LIN {X 0,Y 614.907,Z 968.972,A -85,B 0,C 180,E1 -6595.187,E2 -6595.187} C_VEL
LIN {X 0,Y 616.661,Z 950.759,A -85,B 0,C 180,E1 -6596.845,E2 -6596.845} C_VEL
LIN {X 0,Y 618.487,Z 931.255,A -85,B 0,C 180,E1 -6598.379,E2 -6598.379} C_VEL
LIN {X 0,Y 620.297,Z 912.013,A -85,B 0,C 180,E1 -6599.714,E2 -6599.714} C_VEL
LIN {X 0,Y 622.247,Z 890.482,A -85,B 0,C 180,E1 -6600.998,E2 -6600.998} C_VEL
LIN {X 0,Y 623.869,Z 871.366,A -85,B 0,C 180,E1 -6601.985,E2 -6601.985} C_VEL
LIN {X 0,Y 625.724,Z 847.82,A -85,B 0,C 180,E1 -6603.018,E2 -6603.018} C_VEL
LIN {X 0,Y 627.182,Z 825.971,A -85,B 0,C 180,E1 -6603.807,E2 -6603.807} C_VEL
LIN {X 0,Y 628.648,Z 801.827,A -85,B 0,C 180,E1 -6604.51,E2 -6604.51} C_VEL
LIN {X 0,Y 629.71,Z 779.15,A -85,B 0,C 180,E1 -6605.003,E2 -6605.003} C_VEL
LIN {X 0,Y 630.482,Z 755.478,A -85,B 0,C 180,E1 -6605.381,E2 -6605.381} C_VEL
LIN {X 0,Y 634.576,Z 507.829,A -85,B 0,C 180,E1 -6608.538,E2 -6608.538} C_VEL
LIN {X 0,Y 636.13,Z 410.472,A -85,B 0,C 180,E1 -6609.804,E2 -6609.804} C_VEL
LIN {X 0,Y 632.258,Z 394.616,A -85,B 0,C 180,E1 -6610.318,E2 -6610.318} C_VEL
LIN {X 0,Y 620.448,Z 374.384,A -85,B 0,C 180,E1 -6611.533,E2 -6611.533} C_VEL
LIN {X 0,Y 612.728,Z 354.981,A -85,B 0,C 180,E1 -6613.911,E2 -6613.911} C_VEL
LIN {X 0,Y 609.065,Z 345.367,A -85,B 0,C 180,E1 -6615.133,E2 -6615.133} C_VEL
LIN {X 0,Y 609.009,Z 345.37,A -85,B 0,C 180,E1 -6618.07,E2 -6618.07} C_VEL
LIN {X 0,Y 609.077,Z 345.362,A -85,B 0,C 180,E1 -6621.163,E2 -6621.163} C_VEL
LIN {X 0,Y 609.012,Z 345.368,A -85,B 0,C 180,E1 -6624.233,E2 -6624.233} C_VEL
LIN {X 0,Y 609.057,Z 345.366,A -85,B 0,C 180,E1 -6627.42,E2 -6627.42} C_VEL
LIN {X 0,Y 609.014,Z 345.363,A -85,B 0,C 180,E1 -6630.384,E2 -6630.384} C_VEL
LIN {X 0,Y 609.062,Z 345.353,A -85,B 0,C 180,E1 -6633.478,E2 -6633.478} C_VEL
LIN {X 0,Y 609.009,Z 345.353,A -85,B 0,C 180,E1 -6636.384,E2 -6636.384} C_VEL
LIN {X 0,Y 609.076,Z 345.362,A -85,B 0,C 180,E1 -6639.432,E2 -6639.432} C_VEL
LIN {X 0,Y 609.011,Z 345.364,A -85,B 0,C 180,E1 -6642.515,E2 -6642.515} C_VEL
LIN {X 0,Y 609.07,Z 345.348,A -85,B 0,C 180,E1 -6645.647,E2 -6645.647} C_VEL
LIN {X 0,Y 609.012,Z 345.364,A -85,B 0,C 180,E1 -6648.637,E2 -6648.637} C_VEL
LIN {X 0,Y 609.064,Z 345.355,A -85,B 0,C 180,E1 -6651.789,E2 -6651.789} C_VEL
LIN {X 0,Y 609.012,Z 345.356,A -85,B 0,C 180,E1 -6654.725,E2 -6654.725} C_VEL
LIN {X 0,Y 609.069,Z 345.364,A -85,B 0,C 180,E1 -6657.836,E2 -6657.836} C_VEL
LIN {X 0,Y 609.011,Z 345.346,A -85,B 0,C 180,E1 -6660.847,E2 -6660.847} C_VEL
LIN {X 0,Y 609.068,Z 345.363,A -85,B 0,C 180,E1 -6663.954,E2 -6663.954} C_VEL
LIN {X 0,Y 609.014,Z 345.357,A -85,B 0,C 180,E1 -6666.978,E2 -6666.978} C_VEL
LIN {X 0,Y 609.06,Z 345.352,A -85,B 0,C 180,E1 -6670.117,E2 -6670.117} C_VEL
LIN {X 0,Y 609.016,Z 345.364,A -85,B 0,C 180,E1 -6673.095,E2 -6673.095} C_VEL
LIN {X 0,Y 609.062,Z 345.349,A -85,B 0,C 180,E1 -6676.206,E2 -6676.206} C_VEL
LIN {X 0,Y 609.017,Z 345.363,A -85,B 0,C 180,E1 -6679.17,E2 -6679.17} C_VEL
LIN {X 0,Y 609.072,Z 345.357,A -85,B 0,C 180,E1 -6682.286,E2 -6682.286} C_VEL
LIN {X 0,Y 609.013,Z 345.35,A -85,B 0,C 180,E1 -6685.269,E2 -6685.269} C_VEL
LIN {X 0,Y 609.064,Z 345.357,A -85,B 0,C 180,E1 -6688.43,E2 -6688.43} C_VEL
LIN {X 0,Y 609.017,Z 345.366,A -85,B 0,C 180,E1 -6691.379,E2 -6691.379} C_VEL
LIN {X 0,Y 609.065,Z 345.36,A -85,B 0,C 180,E1 -6694.5,E2 -6694.5} C_VEL
LIN {X 0,Y 609.018,Z 345.364,A -85,B 0,C 180,E1 -6697.534,E2 -6697.534} C_VEL
LIN {X 0,Y 609.061,Z 345.36,A -85,B 0,C 180,E1 -6700.674,E2 -6700.674} C_VEL
LIN {X 0,Y 609.015,Z 345.332,A -85,B 0,C 180,E1 -6703.611,E2 -6703.611} C_VEL
LIN {X 0,Y 609.059,Z 345.368,A -85,B 0,C 180,E1 -6706.797,E2 -6706.797} C_VEL
LIN {X 0,Y 609.062,Z 345.576,A -85,B 0,C 180,E1 -6709.113,E2 -6709.113} C_VEL
LIN {X 0,Y 611.013,Z 350.763,A -85,B 0,C 180,E1 -6709.765,E2 -6709.765} C_VEL
LIN {X 0,Y 626.828,Z 375.591,A -85,B 0,C 180,E1 -6711.41,E2 -6711.41} C_VEL
LIN {X 0,Y 636.341,Z 391.797,A -85,B 0,C 180,E1 -6712.363,E2 -6712.363} C_VEL
LIN {X 0,Y 635.973,Z 412.733,A -85,B 0,C 180,E1 -6712.635,E2 -6712.635} C_VEL
LIN {X 0,Y 635.046,Z 420.434,A -85,B 0,C 180,E1 -6712.677,E2 -6712.677} C_VEL
LIN {X 0,Y 629.809,Z 441.007,A -85,B 0,C 180,E1 -6712.587,E2 -6712.587} C_VEL
LIN {X 0,Y 629.133,Z 447.61,A -85,B 0,C 180,E1 -6712.632,E2 -6712.632} C_VEL
LIN {X 0,Y 624.626,Z 698.687,A -85,B 0,C 180,E1 -6715.87,E2 -6715.87} C_VEL
LIN {X 0,Y 623.697,Z 743.497,A -85,B 0,C 180,E1 -6716.476,E2 -6716.476} C_VEL
LIN {X 0,Y 622.627,Z 767.01,A -85,B 0,C 180,E1 -6716.956,E2 -6716.956} C_VEL
LIN {X 0,Y 621.497,Z 787.189,A -85,B 0,C 180,E1 -6717.49,E2 -6717.49} C_VEL
LIN {X 0,Y 619.803,Z 812.008,A -85,B 0,C 180,E1 -6718.324,E2 -6718.324} C_VEL
LIN {X 0,Y 618.178,Z 832.167,A -85,B 0,C 180,E1 -6719.153,E2 -6719.153} C_VEL
LIN {X 0,Y 616.198,Z 855.203,A -85,B 0,C 180,E1 -6720.282,E2 -6720.282} C_VEL
LIN {X 0,Y 614.304,Z 874.686,A -85,B 0,C 180,E1 -6721.41,E2 -6721.41} C_VEL
LIN {X 0,Y 612.292,Z 894.753,A -85,B 0,C 180,E1 -6722.738,E2 -6722.738} C_VEL
LIN {X 0,Y 610.169,Z 914.461,A -85,B 0,C 180,E1 -6724.262,E2 -6724.262} C_VEL
LIN {X 0,Y 608.261,Z 932.973,A -85,B 0,C 180,E1 -6725.89,E2 -6725.89} C_VEL
LIN {X 0,Y 606.372,Z 950.537,A -85,B 0,C 180,E1 -6727.68,E2 -6727.68} C_VEL
LIN {X 0,Y 604.843,Z 966.182,A -85,B 0,C 180,E1 -6729.484,E2 -6729.484} C_VEL
LIN {X 0,Y 603.374,Z 981.698,A -85,B 0,C 180,E1 -6731.548,E2 -6731.548} C_VEL
LIN {X 0,Y 602.275,Z 995.359,A -85,B 0,C 180,E1 -6733.607,E2 -6733.607} C_VEL
LIN {X 0,Y 601.407,Z 1007.51,A -85,B 0,C 180,E1 -6735.764,E2 -6735.764} C_VEL
LIN {X 0,Y 600.8,Z 1017.904,A -85,B 0,C 180,E1 -6737.895,E2 -6737.895} C_VEL
LIN {X 0,Y 600.376,Z 1026.879,A -85,B 0,C 180,E1 -6740.123,E2 -6740.123} C_VEL
LIN {X 0,Y 600.123,Z 1033.674,A -85,B 0,C 180,E1 -6742.148,E2 -6742.148} C_VEL
LIN {X 0,Y 599.975,Z 1040.012,A -85,B 0,C 180,E1 -6744.549,E2 -6744.549} C_VEL
LIN {X 0,Y 599.921,Z 1043.917,A -85,B 0,C 180,E1 -6746.56,E2 -6746.56} C_VEL
LIN {X 0,Y 599.913,Z 1046.869,A -85,B 0,C 180,E1 -6748.758,E2 -6748.758} C_VEL
LIN {X 0,Y 599.909,Z 1048.271,A -85,B 0,C 180,E1 -6751.051,E2 -6751.051} C_VEL
LIN {X 0,Y 599.907,Z 1048.267,A -85,B 0,C 180,E1 -6753.057,E2 -6753.057} C_VEL
LIN {X 0,Y 599.914,Z 1046.729,A -85,B 0,C 180,E1 -6755.452,E2 -6755.452} C_VEL
LIN {X 0,Y 599.92,Z 1043.857,A -85,B 0,C 180,E1 -6757.566,E2 -6757.566} C_VEL
LIN {X 0,Y 599.977,Z 1039.899,A -85,B 0,C 180,E1 -6759.593,E2 -6759.593} C_VEL
LIN {X 0,Y 600.131,Z 1033.43,A -85,B 0,C 180,E1 -6762.021,E2 -6762.021} C_VEL
LIN {X 0,Y 600.376,Z 1026.855,A -85,B 0,C 180,E1 -6763.974,E2 -6763.974} C_VEL
LIN {X 0,Y 600.809,Z 1017.709,A -85,B 0,C 180,E1 -6766.236,E2 -6766.236} C_VEL
LIN {X 0,Y 601.404,Z 1007.563,A -85,B 0,C 180,E1 -6768.314,E2 -6768.314} C_VEL
LIN {X 0,Y 602.235,Z 995.823,A -85,B 0,C 180,E1 -6770.406,E2 -6770.406} C_VEL
LIN {X 0,Y 603.299,Z 982.647,A -85,B 0,C 180,E1 -6772.408,E2 -6772.408} C_VEL
LIN {X 0,Y 604.779,Z 966.914,A -85,B 0,C 180,E1 -6774.518,E2 -6774.518} C_VEL
LIN {X 0,Y 606.352,Z 950.764,A -85,B 0,C 180,E1 -6776.386,E2 -6776.386} C_VEL
LIN {X 0,Y 608.209,Z 933.493,A -85,B 0,C 180,E1 -6778.153,E2 -6778.153} C_VEL
LIN {X 0,Y 610.106,Z 915.133,A -85,B 0,C 180,E1 -6779.774,E2 -6779.774} C_VEL
LIN {X 0,Y 612.122,Z 896.309,A -85,B 0,C 180,E1 -6781.24,E2 -6781.24} C_VEL
LIN {X 0,Y 614.194,Z 875.91,A -85,B 0,C 180,E1 -6782.606,E2 -6782.606} C_VEL
LIN {X 0,Y 615.954,Z 857.768,A -85,B 0,C 180,E1 -6783.667,E2 -6783.667} C_VEL
LIN {X 0,Y 617.994,Z 834.601,A -85,B 0,C 180,E1 -6784.83,E2 -6784.83} C_VEL
LIN {X 0,Y 619.641,Z 814.117,A -85,B 0,C 180,E1 -6785.686,E2 -6785.686} C_VEL
LIN {X 0,Y 621.334,Z 790.192,A -85,B 0,C 180,E1 -6786.514,E2 -6786.514} C_VEL
LIN {X 0,Y 622.573,Z 768.29,A -85,B 0,C 180,E1 -6787.105,E2 -6787.105} C_VEL
LIN {X 0,Y 623.558,Z 746.916,A -85,B 0,C 180,E1 -6787.553,E2 -6787.553} C_VEL
LIN {X 0,Y 624.385,Z 714.088,A -85,B 0,C 180,E1 -6788.027,E2 -6788.027} C_VEL
LIN {X 0,Y 629.115,Z 459.765,A -85,B 0,C 180,E1 -6791.323,E2 -6791.323} C_VEL
LIN {X 0,Y 630.263,Z 394.469,A -85,B 0,C 180,E1 -6792.193,E2 -6792.193} C_VEL
LIN {X 0,Y 616.493,Z 371.695,A -85,B 0,C 180,E1 -6793.666,E2 -6793.666} C_VEL
LIN {X 0,Y 604.629,Z 353.842,A -85,B 0,C 180,E1 -6794.994,E2 -6794.994} C_VEL
LIN {X 0,Y 602.702,Z 350.561,A -85,B 0,C 180,E1 -6795.24,E2 -6795.24} C_VEL
LIN {X 0,Y 601.12,Z 346.347,A -85,B 0,C 180,E1 -6795.859,E2 -6795.859} C_VEL
LIN {X 0,Y 601.072,Z 346.326,A -85,B 0,C 180,E1 -6798.795,E2 -6798.795} C_VEL
LIN {X 0,Y 601.127,Z 346.352,A -85,B 0,C 180,E1 -6801.895,E2 -6801.895} C_VEL
LIN {X 0,Y 601.077,Z 346.322,A -85,B 0,C 180,E1 -6804.977,E2 -6804.977} C_VEL
LIN {X 0,Y 601.104,Z 346.343,A -85,B 0,C 180,E1 -6808.213,E2 -6808.213} C_VEL
LIN {X 0,Y 601.084,Z 346.351,A -85,B 0,C 180,E1 -6811.157,E2 -6811.157} C_VEL
LIN {X 0,Y 601.088,Z 346.344,A -85,B 0,C 180,E1 -6814.479,E2 -6814.479} C_VEL
LIN {X 0,Y 601.096,Z 346.355,A -85,B 0,C 180,E1 -6817.402,E2 -6817.402} C_VEL
LIN {X 0,Y 601.083,Z 346.353,A -85,B 0,C 180,E1 -6820.668,E2 -6820.668} C_VEL
LIN {X 0,Y 601.113,Z 346.353,A -85,B 0,C 180,E1 -6823.695,E2 -6823.695} C_VEL
LIN {X 0,Y 601.078,Z 346.349,A -85,B 0,C 180,E1 -6826.827,E2 -6826.827} C_VEL
LIN {X 0,Y 601.116,Z 346.343,A -85,B 0,C 180,E1 -6829.844,E2 -6829.844} C_VEL
LIN {X 0,Y 601.076,Z 346.352,A -85,B 0,C 180,E1 -6833.025,E2 -6833.025} C_VEL
LIN {X 0,Y 601.13,Z 346.353,A -85,B 0,C 180,E1 -6836.09,E2 -6836.09} C_VEL
LIN {X 0,Y 601.071,Z 346.345,A -85,B 0,C 180,E1 -6839.237,E2 -6839.237} C_VEL
LIN {X 0,Y 601.135,Z 346.339,A -85,B 0,C 180,E1 -6842.288,E2 -6842.288} C_VEL
LIN {X 0,Y 601.072,Z 346.355,A -85,B 0,C 180,E1 -6845.441,E2 -6845.441} C_VEL
LIN {X 0,Y 601.14,Z 346.35,A -85,B 0,C 180,E1 -6848.513,E2 -6848.513} C_VEL
LIN {X 0,Y 601.071,Z 346.34,A -85,B 0,C 180,E1 -6851.612,E2 -6851.612} C_VEL
LIN {X 0,Y 601.132,Z 346.337,A -85,B 0,C 180,E1 -6854.744,E2 -6854.744} C_VEL
LIN {X 0,Y 601.076,Z 346.355,A -85,B 0,C 180,E1 -6857.823,E2 -6857.823} C_VEL
LIN {X 0,Y 601.107,Z 346.352,A -85,B 0,C 180,E1 -6861.065,E2 -6861.065} C_VEL
LIN {X 0,Y 601.074,Z 346.344,A -85,B 0,C 180,E1 -6863.947,E2 -6863.947} C_VEL
LIN {X 0,Y 601.108,Z 346.341,A -85,B 0,C 180,E1 -6867.136,E2 -6867.136} C_VEL
LIN {X 0,Y 601.078,Z 346.354,A -85,B 0,C 180,E1 -6870.047,E2 -6870.047} C_VEL
LIN {X 0,Y 601.103,Z 346.355,A -85,B 0,C 180,E1 -6873.294,E2 -6873.294} C_VEL
LIN {X 0,Y 601.079,Z 346.357,A -85,B 0,C 180,E1 -6876.216,E2 -6876.216} C_VEL
LIN {X 0,Y 601.093,Z 346.355,A -85,B 0,C 180,E1 -6879.48,E2 -6879.48} C_VEL
LIN {X 0,Y 601.079,Z 346.346,A -85,B 0,C 180,E1 -6882.355,E2 -6882.355} C_VEL
LIN {X 0,Y 601.088,Z 346.48,A -85,B 0,C 180,E1 -6883.997,E2 -6883.997} C_VEL
LIN {X 0,Y 602.408,Z 349.863,A -85,B 0,C 180,E1 -6884.463,E2 -6884.463} C_VEL
LIN {X 0,Y 610.096,Z 368.505,A -85,B 0,C 180,E1 -6886.967,E2 -6886.967} C_VEL
LIN {X 0,Y 612.618,Z 374.622,A -85,B 0,C 180,E1 -6887.713,E2 -6887.713} C_VEL
LIN {X 0,Y 626.907,Z 398.785,A -85,B 0,C 180,E1 -6889.271,E2 -6889.271} C_VEL
LIN {X 0,Y 630.302,Z 413.187,A -85,B 0,C 180,E1 -6889.753,E2 -6889.753} C_VEL
LIN {X 0,Y 625.305,Z 678.851,A -85,B 0,C 180,E1 -6893.209,E2 -6893.209} C_VEL
LIN {X 0,Y 623.609,Z 766.876,A -85,B 0,C 180,E1 -6894.36,E2 -6894.36} C_VEL
LIN {X 0,Y 622.513,Z 792.116,A -85,B 0,C 180,E1 -6894.847,E2 -6894.847} C_VEL
LIN {X 0,Y 621.327,Z 812.813,A -85,B 0,C 180,E1 -6895.38,E2 -6895.38} C_VEL
LIN {X 0,Y 619.815,Z 835.949,A -85,B 0,C 180,E1 -6896.126,E2 -6896.126} C_VEL
LIN {X 0,Y 618.029,Z 858.133,A -85,B 0,C 180,E1 -6897.015,E2 -6897.015} C_VEL
LIN {X 0,Y 616.219,Z 879.499,A -85,B 0,C 180,E1 -6898.026,E2 -6898.026} C_VEL
LIN {X 0,Y 614.165,Z 901.367,A -85,B 0,C 180,E1 -6899.256,E2 -6899.256} C_VEL
LIN {X 0,Y 612.36,Z 919.919,A -85,B 0,C 180,E1 -6900.454,E2 -6900.454} C_VEL
LIN {X 0,Y 610.169,Z 941.37,A -85,B 0,C 180,E1 -6902.052,E2 -6902.052} C_VEL
LIN {X 0,Y 608.466,Z 958.204,A -85,B 0,C 180,E1 -6903.488,E2 -6903.488} C_VEL
LIN {X 0,Y 606.561,Z 977.386,A -85,B 0,C 180,E1 -6905.351,E2 -6905.351} C_VEL
LIN {X 0,Y 605.093,Z 992.65,A -85,B 0,C 180,E1 -6907.047,E2 -6907.047} C_VEL
LIN {X 0,Y 603.751,Z 1007.707,A -85,B 0,C 180,E1 -6908.938,E2 -6908.938} C_VEL
LIN {X 0,Y 602.589,Z 1021.238,A -85,B 0,C 180,E1 -6910.92,E2 -6910.92} C_VEL
LIN {X 0,Y 601.668,Z 1033.688,A -85,B 0,C 180,E1 -6912.993,E2 -6912.993} C_VEL
LIN {X 0,Y 600.962,Z 1044.707,A -85,B 0,C 180,E1 -6915.168,E2 -6915.168} C_VEL
LIN {X 0,Y 600.515,Z 1053.583,A -85,B 0,C 180,E1 -6917.206,E2 -6917.206} C_VEL
LIN {X 0,Y 600.189,Z 1061.907,A -85,B 0,C 180,E1 -6919.538,E2 -6919.538} C_VEL
LIN {X 0,Y 600.028,Z 1067.491,A -85,B 0,C 180,E1 -6921.471,E2 -6921.471} C_VEL
LIN {X 0,Y 599.946,Z 1072.695,A -85,B 0,C 180,E1 -6923.781,E2 -6923.781} C_VEL
LIN {X 0,Y 599.911,Z 1076.009,A -85,B 0,C 180,E1 -6925.986,E2 -6925.986} C_VEL
LIN {X 0,Y 599.906,Z 1077.835,A -85,B 0,C 180,E1 -6927.994,E2 -6927.994} C_VEL
LIN {X 0,Y 599.895,Z 1078.417,A -85,B 0,C 180,E1 -6930.382,E2 -6930.382} C_VEL
LIN {X 0,Y 599.908,Z 1077.495,A -85,B 0,C 180,E1 -6932.484,E2 -6932.484} C_VEL
LIN {X 0,Y 599.925,Z 1075.085,A -85,B 0,C 180,E1 -6934.78,E2 -6934.78} C_VEL
LIN {X 0,Y 599.968,Z 1071.102,A -85,B 0,C 180,E1 -6936.988,E2 -6936.988} C_VEL
LIN {X 0,Y 600.05,Z 1066.219,A -85,B 0,C 180,E1 -6939.012,E2 -6939.012} C_VEL
LIN {X 0,Y 600.302,Z 1058.66,A -85,B 0,C 180,E1 -6941.432,E2 -6941.432} C_VEL
LIN {X 0,Y 600.649,Z 1050.747,A -85,B 0,C 180,E1 -6943.477,E2 -6943.477} C_VEL
LIN {X 0,Y 601.23,Z 1040.401,A -85,B 0,C 180,E1 -6945.729,E2 -6945.729} C_VEL
LIN {X 0,Y 601.991,Z 1029.111,A -85,B 0,C 180,E1 -6947.795,E2 -6947.795} C_VEL
LIN {X 0,Y 603.057,Z 1015.705,A -85,B 0,C 180,E1 -6949.93,E2 -6949.93} C_VEL
LIN {X 0,Y 604.209,Z 1002.366,A -85,B 0,C 180,E1 -6951.758,E2 -6951.758} C_VEL
LIN {X 0,Y 605.684,Z 986.675,A -85,B 0,C 180,E1 -6953.65,E2 -6953.65} C_VEL
LIN {X 0,Y 607.335,Z 969.481,A -85,B 0,C 180,E1 -6955.448,E2 -6955.448} C_VEL
LIN {X 0,Y 609.031,Z 952.779,A -85,B 0,C 180,E1 -6956.997,E2 -6956.997} C_VEL
LIN {X 0,Y 611.099,Z 932.382,A -85,B 0,C 180,E1 -6958.647,E2 -6958.647} C_VEL
LIN {X 0,Y 612.926,Z 914.014,A -85,B 0,C 180,E1 -6959.946,E2 -6959.946} C_VEL
LIN {X 0,Y 615.152,Z 891.169,A -85,B 0,C 180,E1 -6961.342,E2 -6961.342} C_VEL
LIN {X 0,Y 616.861,Z 872.159,A -85,B 0,C 180,E1 -6962.338,E2 -6962.338} C_VEL
LIN {X 0,Y 618.757,Z 849.985,A -85,B 0,C 180,E1 -6963.336,E2 -6963.336} C_VEL
LIN {X 0,Y 620.364,Z 827.239,A -85,B 0,C 180,E1 -6964.174,E2 -6964.174} C_VEL
LIN {X 0,Y 621.869,Z 804.051,A -85,B 0,C 180,E1 -6964.869,E2 -6964.869} C_VEL
LIN {X 0,Y 623.087,Z 780.045,A -85,B 0,C 180,E1 -6965.406,E2 -6965.406} C_VEL
LIN {X 0,Y 623.869,Z 757.754,A -85,B 0,C 180,E1 -6965.771,E2 -6965.771} C_VEL
LIN {X 0,Y 628.139,Z 514.362,A -85,B 0,C 180,E1 -6968.903,E2 -6968.903} C_VEL
LIN {X 0,Y 629.865,Z 412.184,A -85,B 0,C 180,E1 -6970.243,E2 -6970.243} C_VEL
LIN {X 0,Y 626.549,Z 398.688,A -85,B 0,C 180,E1 -6970.691,E2 -6970.691} C_VEL
LIN {X 0,Y 612.132,Z 374.17,A -85,B 0,C 180,E1 -6972.202,E2 -6972.202} C_VEL
LIN {X 0,Y 605.013,Z 356.379,A -85,B 0,C 180,E1 -6974.442,E2 -6974.442} C_VEL
LIN {X 0,Y 602.095,Z 349.342,A -85,B 0,C 180,E1 -6975.374,E2 -6975.374} C_VEL
LIN {X 0,Y 601.073,Z 346.362,A -85,B 0,C 180,E1 -6975.782,E2 -6975.782} C_VEL
LIN {X 0,Y 601.141,Z 346.354,A -85,B 0,C 180,E1 -6978.893,E2 -6978.893} C_VEL
LIN {X 0,Y 601.072,Z 346.354,A -85,B 0,C 180,E1 -6982.012,E2 -6982.012} C_VEL
LIN {X 0,Y 601.137,Z 346.344,A -85,B 0,C 180,E1 -6985.097,E2 -6985.097} C_VEL
LIN {X 0,Y 601.07,Z 346.351,A -85,B 0,C 180,E1 -6988.174,E2 -6988.174} C_VEL
LIN {X 0,Y 601.146,Z 346.349,A -85,B 0,C 180,E1 -6991.269,E2 -6991.269} C_VEL
LIN {X 0,Y 601.073,Z 346.353,A -85,B 0,C 180,E1 -6994.373,E2 -6994.373} C_VEL
LIN {X 0,Y 601.128,Z 346.34,A -85,B 0,C 180,E1 -6997.507,E2 -6997.507} C_VEL
LIN {X 0,Y 601.071,Z 346.344,A -85,B 0,C 180,E1 -7000.466,E2 -7000.466} C_VEL
LIN {X 0,Y 601.132,Z 346.354,A -85,B 0,C 180,E1 -7003.574,E2 -7003.574} C_VEL
LIN {X 0,Y 601.071,Z 346.348,A -85,B 0,C 180,E1 -7006.533,E2 -7006.533} C_VEL
LIN {X 0,Y 601.13,Z 346.339,A -85,B 0,C 180,E1 -7009.651,E2 -7009.651} C_VEL
LIN {X 0,Y 601.073,Z 346.354,A -85,B 0,C 180,E1 -7012.641,E2 -7012.641} C_VEL
LIN {X 0,Y 601.132,Z 346.334,A -85,B 0,C 180,E1 -7015.707,E2 -7015.707} C_VEL
LIN {X 0,Y 601.073,Z 346.353,A -85,B 0,C 180,E1 -7018.763,E2 -7018.763} C_VEL
LIN {X 0,Y 601.129,Z 346.339,A -85,B 0,C 180,E1 -7021.906,E2 -7021.906} C_VEL
LIN {X 0,Y 601.075,Z 346.346,A -85,B 0,C 180,E1 -7024.962,E2 -7024.962} C_VEL
LIN {X 0,Y 601.119,Z 346.354,A -85,B 0,C 180,E1 -7028.128,E2 -7028.128} C_VEL
LIN {X 0,Y 601.077,Z 346.335,A -85,B 0,C 180,E1 -7031.126,E2 -7031.126} C_VEL
LIN {X 0,Y 601.106,Z 346.351,A -85,B 0,C 180,E1 -7034.35,E2 -7034.35} C_VEL
LIN {X 0,Y 601.084,Z 346.347,A -85,B 0,C 180,E1 -7037.323,E2 -7037.323} C_VEL
LIN {X 0,Y 601.087,Z 346.339,A -85,B 0,C 180,E1 -7040.65,E2 -7040.65} C_VEL
LIN {X 0,Y 601.096,Z 346.353,A -85,B 0,C 180,E1 -7043.572,E2 -7043.572} C_VEL
LIN {X 0,Y 601.088,Z 346.357,A -85,B 0,C 180,E1 -7046.795,E2 -7046.795} C_VEL
LIN {X 0,Y 601.101,Z 346.337,A -85,B 0,C 180,E1 -7049.737,E2 -7049.737} C_VEL
LIN {X 0,Y 601.083,Z 346.343,A -85,B 0,C 180,E1 -7052.954,E2 -7052.954} C_VEL
LIN {X 0,Y 601.115,Z 346.351,A -85,B 0,C 180,E1 -7055.957,E2 -7055.957} C_VEL
LIN {X 0,Y 601.079,Z 346.351,A -85,B 0,C 180,E1 -7059.178,E2 -7059.178} C_VEL
LIN {X 0,Y 601.133,Z 346.345,A -85,B 0,C 180,E1 -7062.221,E2 -7062.221} C_VEL
LIN {X 0,Y 601.073,Z 346.328,A -85,B 0,C 180,E1 -7065.397,E2 -7065.397} C_VEL
LIN {X 0,Y 601.153,Z 346.432,A -85,B 0,C 180,E1 -7068.487,E2 -7068.487} C_VEL
LIN {X 0,Y 602.862,Z 351.065,A -85,B 0,C 180,E1 -7069.076,E2 -7069.076} C_VEL
LIN {X 0,Y 616.619,Z 372.529,A -85,B 0,C 180,E1 -7070.559,E2 -7070.559} C_VEL
LIN {X 0,Y 630.095,Z 394.837,A -85,B 0,C 180,E1 -7071.941,E2 -7071.941} C_VEL
LIN {X 0,Y 629.133,Z 447.61,A -85,B 0,C 180,E1 -7072.632,E2 -7072.632} C_VEL
LIN {X 0,Y 628.244,Z 455.305,A -85,B 0,C 180,E1 -7072.677,E2 -7072.677} C_VEL
LIN {X 0,Y 622.959,Z 475.868,A -85,B 0,C 180,E1 -7072.583,E2 -7072.583} C_VEL
LIN {X 0,Y 622.23,Z 482.476,A -85,B 0,C 180,E1 -7072.624,E2 -7072.624} C_VEL
LIN {X 0,Y 617.517,Z 731.007,A -85,B 0,C 180,E1 -7075.856,E2 -7075.856} C_VEL
LIN {X 0,Y 616.722,Z 753.294,A -85,B 0,C 180,E1 -7076.227,E2 -7076.227} C_VEL
LIN {X 0,Y 615.459,Z 777.86,A -85,B 0,C 180,E1 -7076.792,E2 -7076.792} C_VEL
LIN {X 0,Y 614.004,Z 799.911,A -85,B 0,C 180,E1 -7077.466,E2 -7077.466} C_VEL
LIN {X 0,Y 612.299,Z 822.879,A -85,B 0,C 180,E1 -7078.325,E2 -7078.325} C_VEL
LIN {X 0,Y 610.303,Z 844.777,A -85,B 0,C 180,E1 -7079.332,E2 -7079.332} C_VEL
LIN {X 0,Y 608.392,Z 864.519,A -85,B 0,C 180,E1 -7080.391,E2 -7080.391} C_VEL
LIN {X 0,Y 606.038,Z 886.679,A -85,B 0,C 180,E1 -7081.786,E2 -7081.786} C_VEL
LIN {X 0,Y 604.102,Z 904.459,A -85,B 0,C 180,E1 -7083.077,E2 -7083.077} C_VEL
LIN {X 0,Y 601.738,Z 925.356,A -85,B 0,C 180,E1 -7084.825,E2 -7084.825} C_VEL
LIN {X 0,Y 599.882,Z 941.946,A -85,B 0,C 180,E1 -7086.42,E2 -7086.42} C_VEL
LIN {X 0,Y 597.901,Z 960.025,A -85,B 0,C 180,E1 -7088.413,E2 -7088.413} C_VEL
LIN {X 0,Y 596.425,Z 974.226,A -85,B 0,C 180,E1 -7090.206,E2 -7090.206} C_VEL
LIN {X 0,Y 594.973,Z 989.307,A -85,B 0,C 180,E1 -7092.392,E2 -7092.392} C_VEL
LIN {X 0,Y 593.962,Z 1001.792,A -85,B 0,C 180,E1 -7094.475,E2 -7094.475} C_VEL
LIN {X 0,Y 593.142,Z 1013.486,A -85,B 0,C 180,E1 -7096.746,E2 -7096.746} C_VEL
LIN {X 0,Y 592.636,Z 1022.096,A -85,B 0,C 180,E1 -7098.714,E2 -7098.714} C_VEL
LIN {X 0,Y 592.261,Z 1030.49,A -85,B 0,C 180,E1 -7100.982,E2 -7100.982} C_VEL
LIN {X 0,Y 592.049,Z 1036.745,A -85,B 0,C 180,E1 -7103.113,E2 -7103.113} C_VEL
LIN {X 0,Y 591.963,Z 1041.511,A -85,B 0,C 180,E1 -7105.155,E2 -7105.155} C_VEL
LIN {X 0,Y 591.923,Z 1045.542,A -85,B 0,C 180,E1 -7107.58,E2 -7107.58} C_VEL
LIN {X 0,Y 591.905,Z 1047.554,A -85,B 0,C 180,E1 -7109.613,E2 -7109.613} C_VEL
LIN {X 0,Y 591.896,Z 1048.437,A -85,B 0,C 180,E1 -7111.742,E2 -7111.742} C_VEL
LIN {X 0,Y 591.913,Z 1047.773,A -85,B 0,C 180,E1 -7114.166,E2 -7114.166} C_VEL
LIN {X 0,Y 591.922,Z 1045.899,A -85,B 0,C 180,E1 -7116.206,E2 -7116.206} C_VEL
LIN {X 0,Y 591.95,Z 1042.329,A -85,B 0,C 180,E1 -7118.548,E2 -7118.548} C_VEL
LIN {X 0,Y 592.038,Z 1037.192,A -85,B 0,C 180,E1 -7120.805,E2 -7120.805} C_VEL
LIN {X 0,Y 592.239,Z 1031.206,A -85,B 0,C 180,E1 -7122.877,E2 -7122.877} C_VEL
LIN {X 0,Y 592.617,Z 1022.571,A -85,B 0,C 180,E1 -7125.261,E2 -7125.261} C_VEL
LIN {X 0,Y 593.118,Z 1013.869,A -85,B 0,C 180,E1 -7127.26,E2 -7127.26} C_VEL
LIN {X 0,Y 593.945,Z 1002.028,A -85,B 0,C 180,E1 -7129.573,E2 -7129.573} C_VEL
LIN {X 0,Y 594.974,Z 989.301,A -85,B 0,C 180,E1 -7131.699,E2 -7131.699} C_VEL
LIN {X 0,Y 596.458,Z 973.859,A -85,B 0,C 180,E1 -7133.934,E2 -7133.934} C_VEL
LIN {X 0,Y 597.891,Z 960.118,A -85,B 0,C 180,E1 -7135.667,E2 -7135.667} C_VEL
LIN {X 0,Y 599.873,Z 942.069,A -85,B 0,C 180,E1 -7137.659,E2 -7137.659} C_VEL
LIN {X 0,Y 601.647,Z 926.152,A -85,B 0,C 180,E1 -7139.194,E2 -7139.194} C_VEL
LIN {X 0,Y 603.862,Z 906.891,A -85,B 0,C 180,E1 -7140.829,E2 -7140.829} C_VEL
LIN {X 0,Y 605.902,Z 888.072,A -85,B 0,C 180,E1 -7142.21,E2 -7142.21} C_VEL
LIN {X 0,Y 608.117,Z 867.448,A -85,B 0,C 180,E1 -7143.536,E2 -7143.536} C_VEL
LIN {X 0,Y 610.217,Z 845.785,A -85,B 0,C 180,E1 -7144.709,E2 -7144.709} C_VEL
LIN {X 0,Y 612.113,Z 825.036,A -85,B 0,C 180,E1 -7145.673,E2 -7145.673} C_VEL
LIN {X 0,Y 613.912,Z 801.822,A -85,B 0,C 180,E1 -7146.563,E2 -7146.563} C_VEL
LIN {X 0,Y 615.308,Z 781.023,A -85,B 0,C 180,E1 -7147.213,E2 -7147.213} C_VEL
LIN {X 0,Y 616.707,Z 754.929,A -85,B 0,C 180,E1 -7147.84,E2 -7147.84} C_VEL
LIN {X 0,Y 617.54,Z 732.814,A -85,B 0,C 180,E1 -7148.218,E2 -7148.218} C_VEL
LIN {X 0,Y 622.498,Z 483.595,A -85,B 0,C 180,E1 -7151.483,E2 -7151.483} C_VEL
LIN {X 0,Y 624.172,Z 397.807,A -85,B 0,C 180,E1 -7152.63,E2 -7152.63} C_VEL
LIN {X 0,Y 611.713,Z 377.111,A -85,B 0,C 180,E1 -7153.993,E2 -7153.993} C_VEL
LIN {X 0,Y 600.335,Z 359.822,A -85,B 0,C 180,E1 -7155.292,E2 -7155.292} C_VEL
LIN {X 0,Y 594.515,Z 350.884,A -85,B 0,C 180,E1 -7156.004,E2 -7156.004} C_VEL
LIN {X 0,Y 593.137,Z 347.34,A -85,B 0,C 180,E1 -7156.544,E2 -7156.544} C_VEL
LIN {X 0,Y 593.201,Z 347.303,A -85,B 0,C 180,E1 -7159.664,E2 -7159.664} C_VEL
LIN {X 0,Y 593.135,Z 347.329,A -85,B 0,C 180,E1 -7162.757,E2 -7162.757} C_VEL
LIN {X 0,Y 593.186,Z 347.326,A -85,B 0,C 180,E1 -7165.97,E2 -7165.97} C_VEL
LIN {X 0,Y 593.138,Z 347.336,A -85,B 0,C 180,E1 -7168.946,E2 -7168.946} C_VEL
LIN {X 0,Y 593.191,Z 347.334,A -85,B 0,C 180,E1 -7172.056,E2 -7172.056} C_VEL
LIN {X 0,Y 593.139,Z 347.334,A -85,B 0,C 180,E1 -7175.086,E2 -7175.086} C_VEL
LIN {X 0,Y 593.169,Z 347.33,A -85,B 0,C 180,E1 -7178.336,E2 -7178.336} C_VEL
LIN {X 0,Y 593.146,Z 347.342,A -85,B 0,C 180,E1 -7181.331,E2 -7181.331} C_VEL
LIN {X 0,Y 593.148,Z 347.34,A -85,B 0,C 180,E1 -7184.653,E2 -7184.653} C_VEL
LIN {X 0,Y 593.152,Z 347.341,A -85,B 0,C 180,E1 -7187.539,E2 -7187.539} C_VEL
LIN {X 0,Y 593.14,Z 347.337,A -85,B 0,C 180,E1 -7190.882,E2 -7190.882} C_VEL
LIN {X 0,Y 593.166,Z 347.334,A -85,B 0,C 180,E1 -7193.807,E2 -7193.807} C_VEL
LIN {X 0,Y 593.139,Z 347.342,A -85,B 0,C 180,E1 -7197.004,E2 -7197.004} C_VEL
LIN {X 0,Y 593.177,Z 347.337,A -85,B 0,C 180,E1 -7200,E2 -7200} C_VEL
LIN {X 0,Y 593.135,Z 347.331,A -85,B 0,C 180,E1 -7203.189,E2 -7203.189} C_VEL
LIN {X 0,Y 593.195,Z 347.329,A -85,B 0,C 180,E1 -7206.29,E2 -7206.29} C_VEL
LIN {X 0,Y 593.134,Z 347.344,A -85,B 0,C 180,E1 -7209.411,E2 -7209.411} C_VEL
LIN {X 0,Y 593.199,Z 347.336,A -85,B 0,C 180,E1 -7212.59,E2 -7212.59} C_VEL
LIN {X 0,Y 593.131,Z 347.329,A -85,B 0,C 180,E1 -7215.648,E2 -7215.648} C_VEL
LIN {X 0,Y 593.191,Z 347.325,A -85,B 0,C 180,E1 -7218.781,E2 -7218.781} C_VEL
LIN {X 0,Y 593.135,Z 347.345,A -85,B 0,C 180,E1 -7221.873,E2 -7221.873} C_VEL
LIN {X 0,Y 593.178,Z 347.341,A -85,B 0,C 180,E1 -7225.03,E2 -7225.03} C_VEL
LIN {X 0,Y 593.139,Z 347.339,A -85,B 0,C 180,E1 -7228.056,E2 -7228.056} C_VEL
LIN {X 0,Y 593.16,Z 347.342,A -85,B 0,C 180,E1 -7231.279,E2 -7231.279} C_VEL
LIN {X 0,Y 593.146,Z 347.348,A -85,B 0,C 180,E1 -7234.266,E2 -7234.266} C_VEL
LIN {X 0,Y 593.142,Z 347.343,A -85,B 0,C 180,E1 -7237.607,E2 -7237.607} C_VEL
LIN {X 0,Y 593.157,Z 347.344,A -85,B 0,C 180,E1 -7240.513,E2 -7240.513} C_VEL
LIN {X 0,Y 593.203,Z 347.514,A -85,B 0,C 180,E1 -7243.317,E2 -7243.317} C_VEL
LIN {X 0,Y 594.313,Z 350.62,A -85,B 0,C 180,E1 -7243.748,E2 -7243.748} C_VEL
LIN {X 0,Y 599.743,Z 363.46,A -85,B 0,C 180,E1 -7245.555,E2 -7245.555} C_VEL
LIN {X 0,Y 604.178,Z 374.241,A -85,B 0,C 180,E1 -7246.96,E2 -7246.96} C_VEL
LIN {X 0,Y 615.048,Z 392.088,A -85,B 0,C 180,E1 -7248.193,E2 -7248.193} C_VEL
LIN {X 0,Y 621.799,Z 403.971,A -85,B 0,C 180,E1 -7248.937,E2 -7248.937} C_VEL
LIN {X 0,Y 624.187,Z 415.618,A -85,B 0,C 180,E1 -7249.305,E2 -7249.305} C_VEL
LIN {X 0,Y 618.894,Z 680.404,A -85,B 0,C 180,E1 -7252.782,E2 -7252.782} C_VEL
LIN {X 0,Y 617.125,Z 766.737,A -85,B 0,C 180,E1 -7253.923,E2 -7253.923} C_VEL
LIN {X 0,Y 615.96,Z 791.941,A -85,B 0,C 180,E1 -7254.413,E2 -7254.413} C_VEL
LIN {X 0,Y 614.692,Z 812.825,A -85,B 0,C 180,E1 -7254.956,E2 -7254.956} C_VEL
LIN {X 0,Y 612.984,Z 837.056,A -85,B 0,C 180,E1 -7255.753,E2 -7255.753} C_VEL
LIN {X 0,Y 611.217,Z 857.916,A -85,B 0,C 180,E1 -7256.6,E2 -7256.6} C_VEL
LIN {X 0,Y 609.321,Z 878.967,A -85,B 0,C 180,E1 -7257.603,E2 -7257.603} C_VEL
LIN {X 0,Y 607.109,Z 901.141,A -85,B 0,C 180,E1 -7258.859,E2 -7258.859} C_VEL
LIN {X 0,Y 605.152,Z 920.171,A -85,B 0,C 180,E1 -7260.102,E2 -7260.102} C_VEL
LIN {X 0,Y 602.881,Z 941.145,A -85,B 0,C 180,E1 -7261.684,E2 -7261.684} C_VEL
LIN {X 0,Y 601.038,Z 958.14,A -85,B 0,C 180,E1 -7263.149,E2 -7263.149} C_VEL
LIN {X 0,Y 599.032,Z 977.16,A -85,B 0,C 180,E1 -7265.02,E2 -7265.02} C_VEL
LIN {X 0,Y 597.458,Z 992.425,A -85,B 0,C 180,E1 -7266.736,E2 -7266.736} C_VEL
LIN {X 0,Y 595.961,Z 1008.237,A -85,B 0,C 180,E1 -7268.752,E2 -7268.752} C_VEL
LIN {X 0,Y 594.797,Z 1021.223,A -85,B 0,C 180,E1 -7270.66,E2 -7270.66} C_VEL
LIN {X 0,Y 593.816,Z 1033.688,A -85,B 0,C 180,E1 -7272.761,E2 -7272.761} C_VEL
LIN {X 0,Y 593.06,Z 1044.637,A -85,B 0,C 180,E1 -7274.951,E2 -7274.951} C_VEL
LIN {X 0,Y 592.57,Z 1053.582,A -85,B 0,C 180,E1 -7277.031,E2 -7277.031} C_VEL
LIN {X 0,Y 592.22,Z 1061.907,A -85,B 0,C 180,E1 -7279.395,E2 -7279.395} C_VEL
LIN {X 0,Y 592.033,Z 1067.745,A -85,B 0,C 180,E1 -7281.453,E2 -7281.453} C_VEL
LIN {X 0,Y 591.947,Z 1073.015,A -85,B 0,C 180,E1 -7283.891,E2 -7283.891} C_VEL
LIN {X 0,Y 591.912,Z 1076.008,A -85,B 0,C 180,E1 -7285.932,E2 -7285.932} C_VEL
LIN {X 0,Y 591.907,Z 1077.835,A -85,B 0,C 180,E1 -7287.967,E2 -7287.967} C_VEL
LIN {X 0,Y 591.895,Z 1078.417,A -85,B 0,C 180,E1 -7290.387,E2 -7290.387} C_VEL
LIN {X 0,Y 591.907,Z 1077.494,A -85,B 0,C 180,E1 -7292.517,E2 -7292.517} C_VEL
LIN {X 0,Y 591.928,Z 1075.085,A -85,B 0,C 180,E1 -7294.845,E2 -7294.845} C_VEL
LIN {X 0,Y 591.98,Z 1071.102,A -85,B 0,C 180,E1 -7297.083,E2 -7297.083} C_VEL
LIN {X 0,Y 592.069,Z 1066.219,A -85,B 0,C 180,E1 -7299.134,E2 -7299.134} C_VEL
LIN {X 0,Y 592.341,Z 1058.659,A -85,B 0,C 180,E1 -7301.588,E2 -7301.588} C_VEL
LIN {X 0,Y 592.713,Z 1050.747,A -85,B 0,C 180,E1 -7303.661,E2 -7303.661} C_VEL
LIN {X 0,Y 593.342,Z 1040.4,A -85,B 0,C 180,E1 -7305.943,E2 -7305.943} C_VEL
LIN {X 0,Y 594.115,Z 1029.683,A -85,B 0,C 180,E1 -7307.938,E2 -7307.938} C_VEL
LIN {X 0,Y 595.078,Z 1018.012,A -85,B 0,C 180,E1 -7309.841,E2 -7309.841} C_VEL
LIN {X 0,Y 596.44,Z 1002.925,A -85,B 0,C 180,E1 -7311.953,E2 -7311.953} C_VEL
LIN {X 0,Y 597.812,Z 989.017,A -85,B 0,C 180,E1 -7313.667,E2 -7313.667} C_VEL
LIN {X 0,Y 599.748,Z 970.285,A -85,B 0,C 180,E1 -7315.688,E2 -7315.688} C_VEL
LIN {X 0,Y 601.538,Z 953.68,A -85,B 0,C 180,E1 -7317.254,E2 -7317.254} C_VEL
LIN {X 0,Y 603.791,Z 932.835,A -85,B 0,C 180,E1 -7318.972,E2 -7318.972} C_VEL
LIN {X 0,Y 605.723,Z 914.534,A -85,B 0,C 180,E1 -7320.285,E2 -7320.285} C_VEL
LIN {X 0,Y 608.081,Z 891.856,A -85,B 0,C 180,E1 -7321.693,E2 -7321.693} C_VEL
LIN {X 0,Y 609.97,Z 871.941,A -85,B 0,C 180,E1 -7322.748,E2 -7322.748} C_VEL
LIN {X 0,Y 611.957,Z 849.956,A -85,B 0,C 180,E1 -7323.747,E2 -7323.747} C_VEL
LIN {X 0,Y 613.666,Z 826.975,A -85,B 0,C 180,E1 -7324.599,E2 -7324.599} C_VEL
LIN {X 0,Y 615.272,Z 803.625,A -85,B 0,C 180,E1 -7325.302,E2 -7325.302} C_VEL
LIN {X 0,Y 616.529,Z 779.786,A -85,B 0,C 180,E1 -7325.836,E2 -7325.836} C_VEL
LIN {X 0,Y 617.343,Z 757.549,A -85,B 0,C 180,E1 -7326.203,E2 -7326.203} C_VEL
LIN {X 0,Y 621.875,Z 513.243,A -85,B 0,C 180,E1 -7329.374,E2 -7329.374} C_VEL
LIN {X 0,Y 623.645,Z 413.984,A -85,B 0,C 180,E1 -7330.689,E2 -7330.689} C_VEL
LIN {X 0,Y 620.948,Z 402.893,A -85,B 0,C 180,E1 -7331.061,E2 -7331.061} C_VEL
LIN {X 0,Y 606.513,Z 378.526,A -85,B 0,C 180,E1 -7332.6,E2 -7332.6} C_VEL
LIN {X 0,Y 603.652,Z 373.695,A -85,B 0,C 180,E1 -7332.934,E2 -7332.934} C_VEL
LIN {X 0,Y 596.249,Z 354.957,A -85,B 0,C 180,E1 -7335.36,E2 -7335.36} C_VEL
LIN {X 0,Y 593.174,Z 347.515,A -85,B 0,C 180,E1 -7336.38,E2 -7336.38} C_VEL
LIN {X 0,Y 593.143,Z 347.338,A -85,B 0,C 180,E1 -7339.659,E2 -7339.659} C_VEL
LIN {X 0,Y 593.154,Z 347.335,A -85,B 0,C 180,E1 -7342.558,E2 -7342.558} C_VEL
LIN {X 0,Y 593.137,Z 347.335,A -85,B 0,C 180,E1 -7345.864,E2 -7345.864} C_VEL
LIN {X 0,Y 593.179,Z 347.329,A -85,B 0,C 180,E1 -7348.905,E2 -7348.905} C_VEL
LIN {X 0,Y 593.135,Z 347.333,A -85,B 0,C 180,E1 -7352.054,E2 -7352.054} C_VEL
LIN {X 0,Y 593.198,Z 347.34,A -85,B 0,C 180,E1 -7355.183,E2 -7355.183} C_VEL
LIN {X 0,Y 593.132,Z 347.344,A -85,B 0,C 180,E1 -7358.259,E2 -7358.259} C_VEL
LIN {X 0,Y 593.196,Z 347.323,A -85,B 0,C 180,E1 -7361.321,E2 -7361.321} C_VEL
LIN {X 0,Y 593.133,Z 347.338,A -85,B 0,C 180,E1 -7364.452,E2 -7364.452} C_VEL
LIN {X 0,Y 593.199,Z 347.337,A -85,B 0,C 180,E1 -7367.54,E2 -7367.54} C_VEL
LIN {X 0,Y 593.134,Z 347.325,A -85,B 0,C 180,E1 -7370.687,E2 -7370.687} C_VEL
LIN {X 0,Y 593.176,Z 347.337,A -85,B 0,C 180,E1 -7373.904,E2 -7373.904} C_VEL
LIN {X 0,Y 593.139,Z 347.337,A -85,B 0,C 180,E1 -7376.908,E2 -7376.908} C_VEL
LIN {X 0,Y 593.156,Z 347.324,A -85,B 0,C 180,E1 -7380.193,E2 -7380.193} C_VEL
LIN {X 0,Y 593.152,Z 347.341,A -85,B 0,C 180,E1 -7383.189,E2 -7383.189} C_VEL
LIN {X 0,Y 593.142,Z 347.33,A -85,B 0,C 180,E1 -7386.485,E2 -7386.485} C_VEL
LIN {X 0,Y 593.174,Z 347.34,A -85,B 0,C 180,E1 -7389.509,E2 -7389.509} C_VEL
LIN {X 0,Y 593.138,Z 347.343,A -85,B 0,C 180,E1 -7392.758,E2 -7392.758} C_VEL
LIN {X 0,Y 593.189,Z 347.326,A -85,B 0,C 180,E1 -7395.747,E2 -7395.747} C_VEL
LIN {X 0,Y 593.138,Z 347.343,A -85,B 0,C 180,E1 -7398.885,E2 -7398.885} C_VEL
LIN {X 0,Y 593.203,Z 347.327,A -85,B 0,C 180,E1 -7402.018,E2 -7402.018} C_VEL
LIN {X 0,Y 593.136,Z 347.327,A -85,B 0,C 180,E1 -7405.142,E2 -7405.142} C_VEL
LIN {X 0,Y 593.203,Z 347.335,A -85,B 0,C 180,E1 -7408.272,E2 -7408.272} C_VEL
LIN {X 0,Y 593.138,Z 347.344,A -85,B 0,C 180,E1 -7411.28,E2 -7411.28} C_VEL
LIN {X 0,Y 593.196,Z 347.333,A -85,B 0,C 180,E1 -7414.38,E2 -7414.38} C_VEL
LIN {X 0,Y 593.139,Z 347.342,A -85,B 0,C 180,E1 -7417.486,E2 -7417.486} C_VEL
LIN {X 0,Y 593.184,Z 347.337,A -85,B 0,C 180,E1 -7420.665,E2 -7420.665} C_VEL
LIN {X 0,Y 593.142,Z 347.303,A -85,B 0,C 180,E1 -7423.722,E2 -7423.722} C_VEL
LIN {X 0,Y 593.154,Z 347.344,A -85,B 0,C 180,E1 -7427.076,E2 -7427.076} C_VEL
LIN {X 0,Y 593.154,Z 347.392,A -85,B 0,C 180,E1 -7427.839,E2 -7427.839} C_VEL
LIN {X 0,Y 594.654,Z 351.038,A -85,B 0,C 180,E1 -7428.349,E2 -7428.349} C_VEL
LIN {X 0,Y 597.659,Z 355.727,A -85,B 0,C 180,E1 -7428.693,E2 -7428.693} C_VEL
LIN {X 0,Y 614.201,Z 381.749,A -85,B 0,C 180,E1 -7430.503,E2 -7430.503} C_VEL
LIN {X 0,Y 623.877,Z 398.119,A -85,B 0,C 180,E1 -7431.514,E2 -7431.514} C_VEL
LIN {X 0,Y 622.23,Z 482.476,A -85,B 0,C 180,E1 -7432.624,E2 -7432.624} C_VEL
LIN {X 0,Y 621.294,Z 490.172,A -85,B 0,C 180,E1 -7432.667,E2 -7432.667} C_VEL
LIN {X 0,Y 616.01,Z 510.726,A -85,B 0,C 180,E1 -7432.571,E2 -7432.571} C_VEL
LIN {X 0,Y 615.282,Z 517.33,A -85,B 0,C 180,E1 -7432.613,E2 -7432.613} C_VEL
LIN {X 0,Y 610.798,Z 738.818,A -85,B 0,C 180,E1 -7435.53,E2 -7435.53} C_VEL
LIN {X 0,Y 609.666,Z 764.83,A -85,B 0,C 180,E1 -7436.034,E2 -7436.034} C_VEL
LIN {X 0,Y 608.431,Z 785.229,A -85,B 0,C 180,E1 -7436.568,E2 -7436.568} C_VEL
LIN {X 0,Y 606.832,Z 808.119,A -85,B 0,C 180,E1 -7437.316,E2 -7437.316} C_VEL
LIN {X 0,Y 604.856,Z 830.468,A -85,B 0,C 180,E1 -7438.23,E2 -7438.23} C_VEL
LIN {X 0,Y 602.904,Z 851.104,A -85,B 0,C 180,E1 -7439.227,E2 -7439.227} C_VEL
LIN {X 0,Y 600.587,Z 872.854,A -85,B 0,C 180,E1 -7440.475,E2 -7440.475} C_VEL
LIN {X 0,Y 598.536,Z 891.142,A -85,B 0,C 180,E1 -7441.689,E2 -7441.689} C_VEL
LIN {X 0,Y 596.051,Z 912.338,A -85,B 0,C 180,E1 -7443.313,E2 -7443.313} C_VEL
LIN {X 0,Y 594.016,Z 929.15,A -85,B 0,C 180,E1 -7444.794,E2 -7444.794} C_VEL
LIN {X 0,Y 591.899,Z 947.25,A -85,B 0,C 180,E1 -7446.61,E2 -7446.61} C_VEL
LIN {X 0,Y 590.061,Z 962.964,A -85,B 0,C 180,E1 -7448.425,E2 -7448.425} C_VEL
LIN {X 0,Y 588.41,Z 978.342,A -85,B 0,C 180,E1 -7450.442,E2 -7450.442} C_VEL
LIN {X 0,Y 587.046,Z 991.568,A -85,B 0,C 180,E1 -7452.454,E2 -7452.454} C_VEL
LIN {X 0,Y 585.976,Z 1003.957,A -85,B 0,C 180,E1 -7454.602,E2 -7454.602} C_VEL
LIN {X 0,Y 585.111,Z 1015.437,A -85,B 0,C 180,E1 -7456.963,E2 -7456.963} C_VEL
LIN {X 0,Y 584.562,Z 1024.976,A -85,B 0,C 180,E1 -7459.255,E2 -7459.255} C_VEL
LIN {X 0,Y 584.217,Z 1032.642,A -85,B 0,C 180,E1 -7461.536,E2 -7461.536} C_VEL
LIN {X 0,Y 584.029,Z 1038.844,A -85,B 0,C 180,E1 -7463.808,E2 -7463.808} C_VEL
LIN {X 0,Y 583.939,Z 1043.53,A -85,B 0,C 180,E1 -7466.171,E2 -7466.171} C_VEL
LIN {X 0,Y 583.916,Z 1046.369,A -85,B 0,C 180,E1 -7468.234,E2 -7468.234} C_VEL
LIN {X 0,Y 583.905,Z 1048.193,A -85,B 0,C 180,E1 -7470.687,E2 -7470.687} C_VEL
LIN {X 0,Y 583.901,Z 1048.322,A -85,B 0,C 180,E1 -7472.847,E2 -7472.847} C_VEL
LIN {X 0,Y 583.907,Z 1047.208,A -85,B 0,C 180,E1 -7475.01,E2 -7475.01} C_VEL
LIN {X 0,Y 583.921,Z 1044.246,A -85,B 0,C 180,E1 -7477.478,E2 -7477.478} C_VEL
LIN {X 0,Y 583.981,Z 1040.488,A -85,B 0,C 180,E1 -7479.519,E2 -7479.519} C_VEL
LIN {X 0,Y 584.138,Z 1034.778,A -85,B 0,C 180,E1 -7481.853,E2 -7481.853} C_VEL
LIN {X 0,Y 584.42,Z 1027.715,A -85,B 0,C 180,E1 -7484.061,E2 -7484.061} C_VEL
LIN {X 0,Y 584.85,Z 1019.591,A -85,B 0,C 180,E1 -7486.181,E2 -7486.181} C_VEL
LIN {X 0,Y 585.612,Z 1008.323,A -85,B 0,C 180,E1 -7488.62,E2 -7488.62} C_VEL
LIN {X 0,Y 586.517,Z 997.396,A -85,B 0,C 180,E1 -7490.664,E2 -7490.664} C_VEL
LIN {X 0,Y 587.799,Z 983.988,A -85,B 0,C 180,E1 -7492.82,E2 -7492.82} C_VEL
LIN {X 0,Y 589.206,Z 970.769,A -85,B 0,C 180,E1 -7494.675,E2 -7494.675} C_VEL
LIN {X 0,Y 591.158,Z 953.447,A -85,B 0,C 180,E1 -7496.793,E2 -7496.793} C_VEL
LIN {X 0,Y 592.998,Z 937.922,A -85,B 0,C 180,E1 -7498.447,E2 -7498.447} C_VEL
LIN {X 0,Y 595.316,Z 918.528,A -85,B 0,C 180,E1 -7500.257,E2 -7500.257} C_VEL
LIN {X 0,Y 597.342,Z 901.341,A -85,B 0,C 180,E1 -7501.653,E2 -7501.653} C_VEL
LIN {X 0,Y 599.727,Z 881.124,A -85,B 0,C 180,E1 -7503.094,E2 -7503.094} C_VEL
LIN {X 0,Y 601.926,Z 860.711,A -85,B 0,C 180,E1 -7504.336,E2 -7504.336} C_VEL
LIN {X 0,Y 604.066,Z 839.682,A -85,B 0,C 180,E1 -7505.446,E2 -7505.446} C_VEL
LIN {X 0,Y 606.1,Z 817.103,A -85,B 0,C 180,E1 -7506.434,E2 -7506.434} C_VEL
LIN {X 0,Y 607.771,Z 795.967,A -85,B 0,C 180,E1 -7507.206,E2 -7507.206} C_VEL
LIN {X 0,Y 609.436,Z 771.119,A -85,B 0,C 180,E1 -7507.921,E2 -7507.921} C_VEL
LIN {X 0,Y 610.501,Z 750.521,A -85,B 0,C 180,E1 -7508.373,E2 -7508.373} C_VEL
LIN {X 0,Y 611.38,Z 724.593,A -85,B 0,C 180,E1 -7508.786,E2 -7508.786} C_VEL
LIN {X 0,Y 616.669,Z 471.349,A -85,B 0,C 180,E1 -7512.128,E2 -7512.128} C_VEL
LIN {X 0,Y 618.093,Z 401.034,A -85,B 0,C 180,E1 -7513.08,E2 -7513.08} C_VEL
LIN {X 0,Y 606.633,Z 382.039,A -85,B 0,C 180,E1 -7514.362,E2 -7514.362} C_VEL
LIN {X 0,Y 596.058,Z 365.802,A -85,B 0,C 180,E1 -7515.594,E2 -7515.594} C_VEL
LIN {X 0,Y 589.397,Z 356.043,A -85,B 0,C 180,E1 -7516.4,E2 -7516.4} C_VEL
LIN {X 0,Y 586.094,Z 351.126,A -85,B 0,C 180,E1 -7516.834,E2 -7516.834} C_VEL
LIN {X 0,Y 585.241,Z 348.333,A -85,B 0,C 180,E1 -7517.278,E2 -7517.278} C_VEL
LIN {X 0,Y 585.198,Z 348.309,A -85,B 0,C 180,E1 -7520.407,E2 -7520.407} C_VEL
LIN {X 0,Y 585.238,Z 348.294,A -85,B 0,C 180,E1 -7523.418,E2 -7523.418} C_VEL
LIN {X 0,Y 585.198,Z 348.333,A -85,B 0,C 180,E1 -7526.62,E2 -7526.62} C_VEL
LIN {X 0,Y 585.268,Z 348.331,A -85,B 0,C 180,E1 -7529.822,E2 -7529.822} C_VEL
LIN {X 0,Y 585.199,Z 348.333,A -85,B 0,C 180,E1 -7532.967,E2 -7532.967} C_VEL
LIN {X 0,Y 585.239,Z 348.331,A -85,B 0,C 180,E1 -7536.221,E2 -7536.221} C_VEL
LIN {X 0,Y 585.201,Z 348.325,A -85,B 0,C 180,E1 -7539.182,E2 -7539.182} C_VEL
LIN {X 0,Y 585.225,Z 348.321,A -85,B 0,C 180,E1 -7542.435,E2 -7542.435} C_VEL
LIN {X 0,Y 585.208,Z 348.326,A -85,B 0,C 180,E1 -7545.453,E2 -7545.453} C_VEL
LIN {X 0,Y 585.207,Z 348.329,A -85,B 0,C 180,E1 -7548.768,E2 -7548.768} C_VEL
LIN {X 0,Y 585.236,Z 348.33,A -85,B 0,C 180,E1 -7551.847,E2 -7551.847} C_VEL
LIN {X 0,Y 585.199,Z 348.324,A -85,B 0,C 180,E1 -7555.001,E2 -7555.001} C_VEL
LIN {X 0,Y 585.252,Z 348.316,A -85,B 0,C 180,E1 -7558.14,E2 -7558.14} C_VEL
LIN {X 0,Y 585.195,Z 348.333,A -85,B 0,C 180,E1 -7561.273,E2 -7561.273} C_VEL
LIN {X 0,Y 585.258,Z 348.329,A -85,B 0,C 180,E1 -7564.409,E2 -7564.409} C_VEL
LIN {X 0,Y 585.192,Z 348.317,A -85,B 0,C 180,E1 -7567.461,E2 -7567.461} C_VEL
LIN {X 0,Y 585.251,Z 348.315,A -85,B 0,C 180,E1 -7570.633,E2 -7570.633} C_VEL
LIN {X 0,Y 585.197,Z 348.334,A -85,B 0,C 180,E1 -7573.739,E2 -7573.739} C_VEL
LIN {X 0,Y 585.229,Z 348.33,A -85,B 0,C 180,E1 -7576.987,E2 -7576.987} C_VEL
LIN {X 0,Y 585.203,Z 348.318,A -85,B 0,C 180,E1 -7579.992,E2 -7579.992} C_VEL
LIN {X 0,Y 585.204,Z 348.317,A -85,B 0,C 180,E1 -7583.353,E2 -7583.353} C_VEL
LIN {X 0,Y 585.229,Z 348.323,A -85,B 0,C 180,E1 -7586.374,E2 -7586.374} C_VEL
LIN {X 0,Y 585.2,Z 348.331,A -85,B 0,C 180,E1 -7589.59,E2 -7589.59} C_VEL
LIN {X 0,Y 585.249,Z 348.331,A -85,B 0,C 180,E1 -7592.676,E2 -7592.676} C_VEL
LIN {X 0,Y 585.194,Z 348.336,A -85,B 0,C 180,E1 -7595.879,E2 -7595.879} C_VEL
LIN {X 0,Y 585.26,Z 348.328,A -85,B 0,C 180,E1 -7599.081,E2 -7599.081} C_VEL
LIN {X 0,Y 585.194,Z 348.326,A -85,B 0,C 180,E1 -7602.136,E2 -7602.136} C_VEL
LIN {X 0,Y 585.223,Z 348.344,A -85,B 0,C 180,E1 -7602.578,E2 -7602.578} C_VEL
LIN {X 0,Y 586.681,Z 351.97,A -85,B 0,C 180,E1 -7603.113,E2 -7603.113} C_VEL
LIN {X 0,Y 593.473,Z 368.351,A -85,B 0,C 180,E1 -7605.453,E2 -7605.453} C_VEL
LIN {X 0,Y 595.931,Z 373.949,A -85,B 0,C 180,E1 -7606.195,E2 -7606.195} C_VEL
LIN {X 0,Y 609.554,Z 396.18,A -85,B 0,C 180,E1 -7607.785,E2 -7607.785} C_VEL
LIN {X 0,Y 616.287,Z 408.139,A -85,B 0,C 180,E1 -7608.545,E2 -7608.545} C_VEL
LIN {X 0,Y 618.126,Z 417.453,A -85,B 0,C 180,E1 -7608.84,E2 -7608.84} C_VEL
LIN {X 0,Y 612.536,Z 681.518,A -85,B 0,C 180,E1 -7612.339,E2 -7612.339} C_VEL
LIN {X 0,Y 610.689,Z 766.523,A -85,B 0,C 180,E1 -7613.474,E2 -7613.474} C_VEL
LIN {X 0,Y 609.446,Z 791.914,A -85,B 0,C 180,E1 -7613.971,E2 -7613.971} C_VEL
LIN {X 0,Y 608.087,Z 813.136,A -85,B 0,C 180,E1 -7614.529,E2 -7614.529} C_VEL
LIN {X 0,Y 606.241,Z 837.672,A -85,B 0,C 180,E1 -7615.35,E2 -7615.35} C_VEL
LIN {X 0,Y 604.447,Z 857.777,A -85,B 0,C 180,E1 -7616.176,E2 -7616.176} C_VEL
LIN {X 0,Y 602.438,Z 878.777,A -85,B 0,C 180,E1 -7617.187,E2 -7617.187} C_VEL
LIN {X 0,Y 600.086,Z 900.917,A -85,B 0,C 180,E1 -7618.453,E2 -7618.453} C_VEL
LIN {X 0,Y 597.986,Z 920.207,A -85,B 0,C 180,E1 -7619.726,E2 -7619.726} C_VEL
LIN {X 0,Y 595.62,Z 940.919,A -85,B 0,C 180,E1 -7621.307,E2 -7621.307} C_VEL
LIN {X 0,Y 593.657,Z 957.901,A -85,B 0,C 180,E1 -7622.787,E2 -7622.787} C_VEL
LIN {X 0,Y 591.447,Z 977.584,A -85,B 0,C 180,E1 -7624.752,E2 -7624.752} C_VEL
LIN {X 0,Y 589.845,Z 992.199,A -85,B 0,C 180,E1 -7626.418,E2 -7626.418} C_VEL
LIN {X 0,Y 588.248,Z 1008.013,A -85,B 0,C 180,E1 -7628.46,E2 -7628.46} C_VEL
LIN {X 0,Y 586.994,Z 1020.999,A -85,B 0,C 180,E1 -7630.393,E2 -7630.393} C_VEL
LIN {X 0,Y 585.964,Z 1033.662,A -85,B 0,C 180,E1 -7632.532,E2 -7632.532} C_VEL
LIN {X 0,Y 585.19,Z 1044.177,A -85,B 0,C 180,E1 -7634.642,E2 -7634.642} C_VEL
LIN {X 0,Y 584.663,Z 1052.897,A -85,B 0,C 180,E1 -7636.683,E2 -7636.683} C_VEL
LIN {X 0,Y 584.256,Z 1061.604,A -85,B 0,C 180,E1 -7639.149,E2 -7639.149} C_VEL
LIN {X 0,Y 584.044,Z 1067.491,A -85,B 0,C 180,E1 -7641.236,E2 -7641.236} C_VEL
LIN {X 0,Y 583.946,Z 1072.695,A -85,B 0,C 180,E1 -7643.61,E2 -7643.61} C_VEL
LIN {X 0,Y 583.915,Z 1075.894,A -85,B 0,C 180,E1 -7645.777,E2 -7645.777} C_VEL
LIN {X 0,Y 583.909,Z 1077.766,A -85,B 0,C 180,E1 -7647.841,E2 -7647.841} C_VEL
LIN {X 0,Y 583.898,Z 1078.439,A -85,B 0,C 180,E1 -7650.294,E2 -7650.294} C_VEL
LIN {X 0,Y 583.908,Z 1077.562,A -85,B 0,C 180,E1 -7652.454,E2 -7652.454} C_VEL
LIN {X 0,Y 583.922,Z 1075.439,A -85,B 0,C 180,E1 -7654.616,E2 -7654.616} C_VEL
LIN {X 0,Y 583.982,Z 1071.308,A -85,B 0,C 180,E1 -7657.081,E2 -7657.081} C_VEL
LIN {X 0,Y 584.077,Z 1066.474,A -85,B 0,C 180,E1 -7659.161,E2 -7659.161} C_VEL
LIN {X 0,Y 584.348,Z 1059.365,A -85,B 0,C 180,E1 -7661.549,E2 -7661.549} C_VEL
LIN {X 0,Y 584.735,Z 1051.556,A -85,B 0,C 180,E1 -7663.649,E2 -7663.649} C_VEL
LIN {X 0,Y 585.357,Z 1041.888,A -85,B 0,C 180,E1 -7665.861,E2 -7665.861} C_VEL
LIN {X 0,Y 586.229,Z 1030.138,A -85,B 0,C 180,E1 -7668.085,E2 -7668.085} C_VEL
LIN {X 0,Y 587.241,Z 1018.436,A -85,B 0,C 180,E1 -7670.013,E2 -7670.013} C_VEL
LIN {X 0,Y 588.68,Z 1003.484,A -85,B 0,C 180,E1 -7672.152,E2 -7672.152} C_VEL
LIN {X 0,Y 590.127,Z 989.651,A -85,B 0,C 180,E1 -7673.888,E2 -7673.888} C_VEL
LIN {X 0,Y 592.068,Z 972.111,A -85,B 0,C 180,E1 -7675.831,E2 -7675.831} C_VEL
LIN {X 0,Y 593.989,Z 955.14,A -85,B 0,C 180,E1 -7677.467,E2 -7677.467} C_VEL
LIN {X 0,Y 596.231,Z 935.921,A -85,B 0,C 180,E1 -7679.105,E2 -7679.105} C_VEL
LIN {X 0,Y 598.376,Z 916.536,A -85,B 0,C 180,E1 -7680.53,E2 -7680.53} C_VEL
LIN {X 0,Y 600.66,Z 896.054,A -85,B 0,C 180,E1 -7681.85,E2 -7681.85} C_VEL
LIN {X 0,Y 602.819,Z 874.727,A -85,B 0,C 180,E1 -7683.016,E2 -7683.016} C_VEL
LIN {X 0,Y 604.633,Z 855.575,A -85,B 0,C 180,E1 -7683.917,E2 -7683.917} C_VEL
LIN {X 0,Y 606.634,Z 831.946,A -85,B 0,C 180,E1 -7684.853,E2 -7684.853} C_VEL
LIN {X 0,Y 608.207,Z 809.82,A -85,B 0,C 180,E1 -7685.555,E2 -7685.555} C_VEL
LIN {X 0,Y 609.71,Z 785.451,A -85,B 0,C 180,E1 -7686.162,E2 -7686.162} C_VEL
LIN {X 0,Y 610.708,Z 761.524,A -85,B 0,C 180,E1 -7686.581,E2 -7686.581} C_VEL
LIN {X 0,Y 615.333,Z 527.23,A -85,B 0,C 180,E1 -7689.656,E2 -7689.656} C_VEL
LIN {X 0,Y 617.477,Z 415.813,A -85,B 0,C 180,E1 -7691.141,E2 -7691.141} C_VEL
LIN {X 0,Y 615.289,Z 406.929,A -85,B 0,C 180,E1 -7691.447,E2 -7691.447} C_VEL
LIN {X 0,Y 601.355,Z 383.428,A -85,B 0,C 180,E1 -7692.961,E2 -7692.961} C_VEL
LIN {X 0,Y 595.404,Z 373.516,A -85,B 0,C 180,E1 -7693.647,E2 -7693.647} C_VEL
LIN {X 0,Y 588.035,Z 355.483,A -85,B 0,C 180,E1 -7696.071,E2 -7696.071} C_VEL
LIN {X 0,Y 585.253,Z 348.332,A -85,B 0,C 180,E1 -7697.098,E2 -7697.098} C_VEL
LIN {X 0,Y 585.194,Z 348.325,A -85,B 0,C 180,E1 -7700.153,E2 -7700.153} C_VEL
LIN {X 0,Y 585.246,Z 348.322,A -85,B 0,C 180,E1 -7703.275,E2 -7703.275} C_VEL
LIN {X 0,Y 585.201,Z 348.327,A -85,B 0,C 180,E1 -7706.386,E2 -7706.386} C_VEL
LIN {X 0,Y 585.212,Z 348.324,A -85,B 0,C 180,E1 -7709.733,E2 -7709.733} C_VEL
LIN {X 0,Y 585.209,Z 348.316,A -85,B 0,C 180,E1 -7712.638,E2 -7712.638} C_VEL
LIN {X 0,Y 585.206,Z 348.32,A -85,B 0,C 180,E1 -7715.898,E2 -7715.898} C_VEL
LIN {X 0,Y 585.211,Z 348.331,A -85,B 0,C 180,E1 -7718.763,E2 -7718.763} C_VEL
LIN {X 0,Y 585.202,Z 348.33,A -85,B 0,C 180,E1 -7722.12,E2 -7722.12} C_VEL
LIN {X 0,Y 585.251,Z 348.314,A -85,B 0,C 180,E1 -7725.239,E2 -7725.239} C_VEL
LIN {X 0,Y 585.197,Z 348.332,A -85,B 0,C 180,E1 -7728.368,E2 -7728.368} C_VEL
LIN {X 0,Y 585.262,Z 348.313,A -85,B 0,C 180,E1 -7731.568,E2 -7731.568} C_VEL
LIN {X 0,Y 585.195,Z 348.322,A -85,B 0,C 180,E1 -7734.608,E2 -7734.608} C_VEL
LIN {X 0,Y 585.25,Z 348.331,A -85,B 0,C 180,E1 -7737.846,E2 -7737.846} C_VEL
LIN {X 0,Y 585.196,Z 348.31,A -85,B 0,C 180,E1 -7740.881,E2 -7740.881} C_VEL
LIN {X 0,Y 585.233,Z 348.328,A -85,B 0,C 180,E1 -7744.115,E2 -7744.115} C_VEL
LIN {X 0,Y 585.206,Z 348.322,A -85,B 0,C 180,E1 -7747.165,E2 -7747.165} C_VEL
LIN {X 0,Y 585.204,Z 348.314,A -85,B 0,C 180,E1 -7750.534,E2 -7750.534} C_VEL
LIN {X 0,Y 585.242,Z 348.329,A -85,B 0,C 180,E1 -7753.637,E2 -7753.637} C_VEL
LIN {X 0,Y 585.199,Z 348.322,A -85,B 0,C 180,E1 -7756.784,E2 -7756.784} C_VEL
LIN {X 0,Y 585.256,Z 348.321,A -85,B 0,C 180,E1 -7759.876,E2 -7759.876} C_VEL
LIN {X 0,Y 585.2,Z 348.333,A -85,B 0,C 180,E1 -7763.034,E2 -7763.034} C_VEL
LIN {X 0,Y 585.259,Z 348.313,A -85,B 0,C 180,E1 -7766.154,E2 -7766.154} C_VEL
LIN {X 0,Y 585.198,Z 348.318,A -85,B 0,C 180,E1 -7769.253,E2 -7769.253} C_VEL
LIN {X 0,Y 585.252,Z 348.321,A -85,B 0,C 180,E1 -7772.443,E2 -7772.443} C_VEL
LIN {X 0,Y 585.207,Z 348.332,A -85,B 0,C 180,E1 -7775.581,E2 -7775.581} C_VEL
LIN {X 0,Y 585.213,Z 348.33,A -85,B 0,C 180,E1 -7778.959,E2 -7778.959} C_VEL
LIN {X 0,Y 585.23,Z 348.332,A -85,B 0,C 180,E1 -7781.994,E2 -7781.994} C_VEL
LIN {X 0,Y 585.199,Z 348.297,A -85,B 0,C 180,E1 -7785.255,E2 -7785.255} C_VEL
LIN {X 0,Y 585.229,Z 348.482,A -85,B 0,C 180,E1 -7787.188,E2 -7787.188} C_VEL
LIN {X 0,Y 586.433,Z 351.703,A -85,B 0,C 180,E1 -7787.604,E2 -7787.604} C_VEL
LIN {X 0,Y 593.873,Z 362.855,A -85,B 0,C 180,E1 -7788.47,E2 -7788.47} C_VEL
LIN {X 0,Y 604.368,Z 379.261,A -85,B 0,C 180,E1 -7789.648,E2 -7789.648} C_VEL
LIN {X 0,Y 617.684,Z 401.085,A -85,B 0,C 180,E1 -7791.073,E2 -7791.073} C_VEL
LIN {X 0,Y 615.282,Z 517.33,A -85,B 0,C 180,E1 -7792.613,E2 -7792.613} C_VEL
LIN {X 0,Y 614.341,Z 525.026,A -85,B 0,C 180,E1 -7792.656,E2 -7792.656} C_VEL
LIN {X 0,Y 609.054,Z 545.579,A -85,B 0,C 180,E1 -7792.559,E2 -7792.559} C_VEL
LIN {X 0,Y 608.331,Z 552.182,A -85,B 0,C 180,E1 -7792.602,E2 -7792.602} C_VEL
LIN {X 0,Y 604.333,Z 739.177,A -85,B 0,C 180,E1 -7795.087,E2 -7795.087} C_VEL
LIN {X 0,Y 603.148,Z 765.149,A -85,B 0,C 180,E1 -7795.595,E2 -7795.595} C_VEL
LIN {X 0,Y 601.853,Z 785.645,A -85,B 0,C 180,E1 -7796.136,E2 -7796.136} C_VEL
LIN {X 0,Y 600.119,Z 809.127,A -85,B 0,C 180,E1 -7796.915,E2 -7796.915} C_VEL
LIN {X 0,Y 598.083,Z 831.195,A -85,B 0,C 180,E1 -7797.827,E2 -7797.827} C_VEL
LIN {X 0,Y 596.041,Z 851.797,A -85,B 0,C 180,E1 -7798.834,E2 -7798.834} C_VEL
LIN {X 0,Y 593.605,Z 873.488,A -85,B 0,C 180,E1 -7800.093,E2 -7800.093} C_VEL
LIN {X 0,Y 591.43,Z 891.995,A -85,B 0,C 180,E1 -7801.335,E2 -7801.335} C_VEL
LIN {X 0,Y 588.808,Z 913.18,A -85,B 0,C 180,E1 -7802.984,E2 -7802.984} C_VEL
LIN {X 0,Y 586.698,Z 929.682,A -85,B 0,C 180,E1 -7804.458,E2 -7804.458} C_VEL
LIN {X 0,Y 584.333,Z 948.637,A -85,B 0,C 180,E1 -7806.396,E2 -7806.396} C_VEL
LIN {X 0,Y 582.508,Z 963.422,A -85,B 0,C 180,E1 -7808.131,E2 -7808.131} C_VEL
LIN {X 0,Y 580.746,Z 978.759,A -85,B 0,C 180,E1 -7810.173,E2 -7810.173} C_VEL
LIN {X 0,Y 579.359,Z 991.345,A -85,B 0,C 180,E1 -7812.109,E2 -7812.109} C_VEL
LIN {X 0,Y 578.223,Z 1003.569,A -85,B 0,C 180,E1 -7814.247,E2 -7814.247} C_VEL
LIN {X 0,Y 577.31,Z 1014.368,A -85,B 0,C 180,E1 -7816.478,E2 -7816.478} C_VEL
LIN {X 0,Y 576.729,Z 1022.773,A -85,B 0,C 180,E1 -7818.499,E2 -7818.499} C_VEL
LIN {X 0,Y 576.277,Z 1031.524,A -85,B 0,C 180,E1 -7821.016,E2 -7821.016} C_VEL
LIN {X 0,Y 576.058,Z 1037.458,A -85,B 0,C 180,E1 -7823.145,E2 -7823.145} C_VEL
LIN {X 0,Y 575.954,Z 1042.62,A -85,B 0,C 180,E1 -7825.519,E2 -7825.519} C_VEL
LIN {X 0,Y 575.921,Z 1045.947,A -85,B 0,C 180,E1 -7827.811,E2 -7827.811} C_VEL
LIN {X 0,Y 575.923,Z 1047.796,A -85,B 0,C 180,E1 -7829.901,E2 -7829.901} C_VEL
LIN {X 0,Y 575.895,Z 1048.429,A -85,B 0,C 180,E1 -7832.388,E2 -7832.388} C_VEL
LIN {X 0,Y 575.904,Z 1047.597,A -85,B 0,C 180,E1 -7834.481,E2 -7834.481} C_VEL
LIN {X 0,Y 575.925,Z 1045.605,A -85,B 0,C 180,E1 -7836.58,E2 -7836.58} C_VEL
LIN {X 0,Y 575.978,Z 1041.588,A -85,B 0,C 180,E1 -7839.089,E2 -7839.089} C_VEL
LIN {X 0,Y 576.085,Z 1036.789,A -85,B 0,C 180,E1 -7841.209,E2 -7841.209} C_VEL
LIN {X 0,Y 576.351,Z 1030.1,A -85,B 0,C 180,E1 -7843.545,E2 -7843.545} C_VEL
LIN {X 0,Y 576.806,Z 1021.575,A -85,B 0,C 180,E1 -7845.896,E2 -7845.896} C_VEL
LIN {X 0,Y 577.502,Z 1011.945,A -85,B 0,C 180,E1 -7848.159,E2 -7848.159} C_VEL
LIN {X 0,Y 578.438,Z 1000.88,A -85,B 0,C 180,E1 -7850.331,E2 -7850.331} C_VEL
LIN {X 0,Y 579.584,Z 989.371,A -85,B 0,C 180,E1 -7852.305,E2 -7852.305} C_VEL
LIN {X 0,Y 581.192,Z 974.619,A -85,B 0,C 180,E1 -7854.495,E2 -7854.495} C_VEL
LIN {X 0,Y 582.82,Z 960.91,A -85,B 0,C 180,E1 -7856.272,E2 -7856.272} C_VEL
LIN {X 0,Y 584.986,Z 943.44,A -85,B 0,C 180,E1 -7858.259,E2 -7858.259} C_VEL
LIN {X 0,Y 587.079,Z 926.87,A -85,B 0,C 180,E1 -7859.898,E2 -7859.898} C_VEL
LIN {X 0,Y 589.511,Z 907.89,A -85,B 0,C 180,E1 -7861.551,E2 -7861.551} C_VEL
LIN {X 0,Y 591.868,Z 888.411,A -85,B 0,C 180,E1 -7863.013,E2 -7863.013} C_VEL
LIN {X 0,Y 594.357,Z 867.821,A -85,B 0,C 180,E1 -7864.362,E2 -7864.362} C_VEL
LIN {X 0,Y 596.576,Z 847.233,A -85,B 0,C 180,E1 -7865.503,E2 -7865.503} C_VEL
LIN {X 0,Y 598.546,Z 827.813,A -85,B 0,C 180,E1 -7866.432,E2 -7866.432} C_VEL
LIN {X 0,Y 600.712,Z 803.148,A -85,B 0,C 180,E1 -7867.412,E2 -7867.412} C_VEL
LIN {X 0,Y 602.28,Z 782.045,A -85,B 0,C 180,E1 -7868.087,E2 -7868.087} C_VEL
LIN {X 0,Y 603.8,Z 756.854,A -85,B 0,C 180,E1 -7868.711,E2 -7868.711} C_VEL
LIN {X 0,Y 604.743,Z 734.357,A -85,B 0,C 180,E1 -7869.107,E2 -7869.107} C_VEL
LIN {X 0,Y 610.255,Z 487.387,A -85,B 0,C 180,E1 -7872.407,E2 -7872.407} C_VEL
LIN {X 0,Y 612.064,Z 404.383,A -85,B 0,C 180,E1 -7873.537,E2 -7873.537} C_VEL
LIN {X 0,Y 601.821,Z 387.309,A -85,B 0,C 180,E1 -7874.709,E2 -7874.709} C_VEL
LIN {X 0,Y 591.561,Z 371.457,A -85,B 0,C 180,E1 -7875.929,E2 -7875.929} C_VEL
LIN {X 0,Y 584.635,Z 361.326,A -85,B 0,C 180,E1 -7876.783,E2 -7876.783} C_VEL
LIN {X 0,Y 577.839,Z 351.31,A -85,B 0,C 180,E1 -7877.691,E2 -7877.691} C_VEL
LIN {X 0,Y 577.29,Z 349.299,A -85,B 0,C 180,E1 -7877.991,E2 -7877.991} C_VEL
LIN {X 0,Y 577.273,Z 349.313,A -85,B 0,C 180,E1 -7881.051,E2 -7881.051} C_VEL
LIN {X 0,Y 577.263,Z 349.277,A -85,B 0,C 180,E1 -7884.409,E2 -7884.409} C_VEL
LIN {X 0,Y 577.31,Z 349.315,A -85,B 0,C 180,E1 -7887.526,E2 -7887.526} C_VEL
LIN {X 0,Y 577.262,Z 349.321,A -85,B 0,C 180,E1 -7890.647,E2 -7890.647} C_VEL
LIN {X 0,Y 577.313,Z 349.316,A -85,B 0,C 180,E1 -7893.68,E2 -7893.68} C_VEL
LIN {X 0,Y 577.259,Z 349.323,A -85,B 0,C 180,E1 -7896.892,E2 -7896.892} C_VEL
LIN {X 0,Y 577.322,Z 349.319,A -85,B 0,C 180,E1 -7900.05,E2 -7900.05} C_VEL
LIN {X 0,Y 577.259,Z 349.317,A -85,B 0,C 180,E1 -7903.186,E2 -7903.186} C_VEL
LIN {X 0,Y 577.301,Z 349.308,A -85,B 0,C 180,E1 -7906.376,E2 -7906.376} C_VEL
LIN {X 0,Y 577.263,Z 349.316,A -85,B 0,C 180,E1 -7909.42,E2 -7909.42} C_VEL
LIN {X 0,Y 577.275,Z 349.318,A -85,B 0,C 180,E1 -7912.736,E2 -7912.736} C_VEL
LIN {X 0,Y 577.277,Z 349.316,A -85,B 0,C 180,E1 -7915.729,E2 -7915.729} C_VEL
LIN {X 0,Y 577.263,Z 349.31,A -85,B 0,C 180,E1 -7919.008,E2 -7919.008} C_VEL
LIN {X 0,Y 577.299,Z 349.31,A -85,B 0,C 180,E1 -7922.03,E2 -7922.03} C_VEL
LIN {X 0,Y 577.258,Z 349.322,A -85,B 0,C 180,E1 -7925.267,E2 -7925.267} C_VEL
LIN {X 0,Y 577.323,Z 349.311,A -85,B 0,C 180,E1 -7928.365,E2 -7928.365} C_VEL
LIN {X 0,Y 577.255,Z 349.305,A -85,B 0,C 180,E1 -7931.591,E2 -7931.591} C_VEL
LIN {X 0,Y 577.312,Z 349.303,A -85,B 0,C 180,E1 -7934.75,E2 -7934.75} C_VEL
LIN {X 0,Y 577.262,Z 349.322,A -85,B 0,C 180,E1 -7937.854,E2 -7937.854} C_VEL
LIN {X 0,Y 577.273,Z 349.32,A -85,B 0,C 180,E1 -7941.224,E2 -7941.224} C_VEL
LIN {X 0,Y 577.269,Z 349.31,A -85,B 0,C 180,E1 -7944.128,E2 -7944.128} C_VEL
LIN {X 0,Y 577.267,Z 349.311,A -85,B 0,C 180,E1 -7947.435,E2 -7947.435} C_VEL
LIN {X 0,Y 577.285,Z 349.322,A -85,B 0,C 180,E1 -7950.394,E2 -7950.394} C_VEL
LIN {X 0,Y 577.261,Z 349.324,A -85,B 0,C 180,E1 -7953.661,E2 -7953.661} C_VEL
LIN {X 0,Y 577.319,Z 349.32,A -85,B 0,C 180,E1 -7956.854,E2 -7956.854} C_VEL
LIN {X 0,Y 577.256,Z 349.327,A -85,B 0,C 180,E1 -7959.988,E2 -7959.988} C_VEL
LIN {X 0,Y 577.26,Z 349.335,A -85,B 0,C 180,E1 -7961.826,E2 -7961.826} C_VEL
LIN {X 0,Y 578.661,Z 352.927,A -85,B 0,C 180,E1 -7962.369,E2 -7962.369} C_VEL
LIN {X 0,Y 585.725,Z 369.544,A -85,B 0,C 180,E1 -7964.832,E2 -7964.832} C_VEL
LIN {X 0,Y 587.445,Z 373.637,A -85,B 0,C 180,E1 -7965.373,E2 -7965.373} C_VEL
LIN {X 0,Y 598.918,Z 391.689,A -85,B 0,C 180,E1 -7966.763,E2 -7966.763} C_VEL
LIN {X 0,Y 610.774,Z 412.128,A -85,B 0,C 180,E1 -7968.14,E2 -7968.14} C_VEL
LIN {X 0,Y 612.108,Z 419.351,A -85,B 0,C 180,E1 -7968.366,E2 -7968.366} C_VEL
LIN {X 0,Y 606.224,Z 682.374,A -85,B 0,C 180,E1 -7971.883,E2 -7971.883} C_VEL
LIN {X 0,Y 604.297,Z 766.416,A -85,B 0,C 180,E1 -7973.016,E2 -7973.016} C_VEL
LIN {X 0,Y 602.985,Z 791.763,A -85,B 0,C 180,E1 -7973.516,E2 -7973.516} C_VEL
LIN {X 0,Y 601.544,Z 813.171,A -85,B 0,C 180,E1 -7974.084,E2 -7974.084} C_VEL
LIN {X 0,Y 599.667,Z 836.921,A -85,B 0,C 180,E1 -7974.882,E2 -7974.882} C_VEL
LIN {X 0,Y 597.684,Z 858.052,A -85,B 0,C 180,E1 -7975.758,E2 -7975.758} C_VEL
LIN {X 0,Y 595.5,Z 879.666,A -85,B 0,C 180,E1 -7976.813,E2 -7976.813} C_VEL
LIN {X 0,Y 593.014,Z 901.561,A -85,B 0,C 180,E1 -7978.089,E2 -7978.089} C_VEL
LIN {X 0,Y 590.645,Z 922.212,A -85,B 0,C 180,E1 -7979.478,E2 -7979.478} C_VEL
LIN {X 0,Y 588.151,Z 942.533,A -85,B 0,C 180,E1 -7981.075,E2 -7981.075} C_VEL
LIN {X 0,Y 585.978,Z 960.488,A -85,B 0,C 180,E1 -7982.677,E2 -7982.677} C_VEL
LIN {X 0,Y 583.805,Z 978.579,A -85,B 0,C 180,E1 -7984.539,E2 -7984.539} C_VEL
LIN {X 0,Y 582.063,Z 993.683,A -85,B 0,C 180,E1 -7986.298,E2 -7986.298} C_VEL
LIN {X 0,Y 580.309,Z 1009.914,A -85,B 0,C 180,E1 -7988.469,E2 -7988.469} C_VEL
LIN {X 0,Y 579.089,Z 1022.06,A -85,B 0,C 180,E1 -7990.324,E2 -7990.324} C_VEL
LIN {X 0,Y 577.919,Z 1035.491,A -85,B 0,C 180,E1 -7992.687,E2 -7992.687} C_VEL
LIN {X 0,Y 577.186,Z 1045.421,A -85,B 0,C 180,E1 -7994.733,E2 -7994.733} C_VEL
LIN {X 0,Y 576.602,Z 1055.128,A -85,B 0,C 180,E1 -7997.074,E2 -7997.074} C_VEL
LIN {X 0,Y 576.249,Z 1062.512,A -85,B 0,C 180,E1 -7999.3,E2 -7999.3} C_VEL
LIN {X 0,Y 576.044,Z 1068.762,A -85,B 0,C 180,E1 -8001.616,E2 -8001.616} C_VEL
LIN {X 0,Y 575.946,Z 1073.493,A -85,B 0,C 180,E1 -8004.021,E2 -8004.021} C_VEL
LIN {X 0,Y 575.91,Z 1076.235,A -85,B 0,C 180,E1 -8006.018,E2 -8006.018} C_VEL
LIN {X 0,Y 575.895,Z 1078.104,A -85,B 0,C 180,E1 -8008.309,E2 -8008.309} C_VEL
LIN {X 0,Y 575.895,Z 1078.371,A -85,B 0,C 180,E1 -8010.597,E2 -8010.597} C_VEL
LIN {X 0,Y 575.907,Z 1077.425,A -85,B 0,C 180,E1 -8012.687,E2 -8012.687} C_VEL
LIN {X 0,Y 575.932,Z 1074.929,A -85,B 0,C 180,E1 -8015.08,E2 -8015.08} C_VEL
LIN {X 0,Y 575.984,Z 1070.895,A -85,B 0,C 180,E1 -8017.381,E2 -8017.381} C_VEL
LIN {X 0,Y 576.125,Z 1065.965,A -85,B 0,C 180,E1 -8019.49,E2 -8019.49} C_VEL
LIN {X 0,Y 576.434,Z 1058.305,A -85,B 0,C 180,E1 -8022.014,E2 -8022.014} C_VEL
LIN {X 0,Y 576.827,Z 1051.101,A -85,B 0,C 180,E1 -8023.942,E2 -8023.942} C_VEL
LIN {X 0,Y 577.499,Z 1041.233,A -85,B 0,C 180,E1 -8026.186,E2 -8026.186} C_VEL
LIN {X 0,Y 578.433,Z 1029.338,A -85,B 0,C 180,E1 -8028.442,E2 -8028.442} C_VEL
LIN {X 0,Y 579.681,Z 1016.287,A -85,B 0,C 180,E1 -8030.602,E2 -8030.602} C_VEL
LIN {X 0,Y 581.178,Z 1001.706,A -85,B 0,C 180,E1 -8032.667,E2 -8032.667} C_VEL
LIN {X 0,Y 582.858,Z 986.869,A -85,B 0,C 180,E1 -8034.529,E2 -8034.529} C_VEL
LIN {X 0,Y 584.909,Z 969.334,A -85,B 0,C 180,E1 -8036.444,E2 -8036.444} C_VEL
LIN {X 0,Y 586.941,Z 952.681,A -85,B 0,C 180,E1 -8038.046,E2 -8038.046} C_VEL
LIN {X 0,Y 589.459,Z 931.724,A -85,B 0,C 180,E1 -8039.802,E2 -8039.802} C_VEL
LIN {X 0,Y 591.662,Z 913.344,A -85,B 0,C 180,E1 -8041.14,E2 -8041.14} C_VEL
LIN {X 0,Y 594.275,Z 890.446,A -85,B 0,C 180,E1 -8042.576,E2 -8042.576} C_VEL
LIN {X 0,Y 596.269,Z 871.373,A -85,B 0,C 180,E1 -8043.599,E2 -8043.599} C_VEL
LIN {X 0,Y 598.459,Z 849.276,A -85,B 0,C 180,E1 -8044.615,E2 -8044.615} C_VEL
LIN {X 0,Y 600.34,Z 826.581,A -85,B 0,C 180,E1 -8045.467,E2 -8045.467} C_VEL
LIN {X 0,Y 602.136,Z 802.945,A -85,B 0,C 180,E1 -8046.185,E2 -8046.185} C_VEL
LIN {X 0,Y 603.49,Z 779.272,A -85,B 0,C 180,E1 -8046.721,E2 -8046.721} C_VEL
LIN {X 0,Y 604.371,Z 757.158,A -85,B 0,C 180,E1 -8047.091,E2 -8047.091} C_VEL
LIN {X 0,Y 609.472,Z 510.586,A -85,B 0,C 180,E1 -8050.349,E2 -8050.349} C_VEL
LIN {X 0,Y 611.336,Z 417.63,A -85,B 0,C 180,E1 -8051.602,E2 -8051.602} C_VEL
LIN {X 0,Y 609.66,Z 410.943,A -85,B 0,C 180,E1 -8051.84,E2 -8051.84} C_VEL
LIN {X 0,Y 594.048,Z 384.607,A -85,B 0,C 180,E1 -8053.581,E2 -8053.581} C_VEL
LIN {X 0,Y 586.872,Z 372.967,A -85,B 0,C 180,E1 -8054.449,E2 -8054.449} C_VEL
LIN {X 0,Y 581.128,Z 359.046,A -85,B 0,C 180,E1 -8056.373,E2 -8056.373} C_VEL
LIN {X 0,Y 578.336,Z 352.395,A -85,B 0,C 180,E1 -8057.333,E2 -8057.333} C_VEL
LIN {X 0,Y 577.259,Z 349.329,A -85,B 0,C 180,E1 -8057.773,E2 -8057.773} C_VEL
LIN {X 0,Y 577.306,Z 349.313,A -85,B 0,C 180,E1 -8060.789,E2 -8060.789} C_VEL
LIN {X 0,Y 577.257,Z 349.326,A -85,B 0,C 180,E1 -8063.989,E2 -8063.989} C_VEL
LIN {X 0,Y 577.321,Z 349.316,A -85,B 0,C 180,E1 -8067.173,E2 -8067.173} C_VEL
LIN {X 0,Y 577.257,Z 349.32,A -85,B 0,C 180,E1 -8070.304,E2 -8070.304} C_VEL
LIN {X 0,Y 577.307,Z 349.305,A -85,B 0,C 180,E1 -8073.458,E2 -8073.458} C_VEL
LIN {X 0,Y 577.259,Z 349.304,A -85,B 0,C 180,E1 -8076.522,E2 -8076.522} C_VEL
LIN {X 0,Y 577.289,Z 349.313,A -85,B 0,C 180,E1 -8079.732,E2 -8079.732} C_VEL
LIN {X 0,Y 577.27,Z 349.318,A -85,B 0,C 180,E1 -8082.771,E2 -8082.771} C_VEL
LIN {X 0,Y 577.263,Z 349.309,A -85,B 0,C 180,E1 -8086.17,E2 -8086.17} C_VEL
LIN {X 0,Y 577.299,Z 349.315,A -85,B 0,C 180,E1 -8089.219,E2 -8089.219} C_VEL
LIN {X 0,Y 577.257,Z 349.323,A -85,B 0,C 180,E1 -8092.435,E2 -8092.435} C_VEL
LIN {X 0,Y 577.314,Z 349.298,A -85,B 0,C 180,E1 -8095.53,E2 -8095.53} C_VEL
LIN {X 0,Y 577.256,Z 349.32,A -85,B 0,C 180,E1 -8098.71,E2 -8098.71} C_VEL
LIN {X 0,Y 577.313,Z 349.302,A -85,B 0,C 180,E1 -8101.886,E2 -8101.886} C_VEL
LIN {X 0,Y 577.26,Z 349.313,A -85,B 0,C 180,E1 -8104.968,E2 -8104.968} C_VEL
LIN {X 0,Y 577.287,Z 349.324,A -85,B 0,C 180,E1 -8108.266,E2 -8108.266} C_VEL
LIN {X 0,Y 577.277,Z 349.297,A -85,B 0,C 180,E1 -8111.375,E2 -8111.375} C_VEL
LIN {X 0,Y 577.265,Z 349.316,A -85,B 0,C 180,E1 -8114.649,E2 -8114.649} C_VEL
LIN {X 0,Y 577.306,Z 349.311,A -85,B 0,C 180,E1 -8117.748,E2 -8117.748} C_VEL
LIN {X 0,Y 577.259,Z 349.304,A -85,B 0,C 180,E1 -8120.905,E2 -8120.905} C_VEL
LIN {X 0,Y 577.322,Z 349.314,A -85,B 0,C 180,E1 -8124.017,E2 -8124.017} C_VEL
LIN {X 0,Y 577.261,Z 349.322,A -85,B 0,C 180,E1 -8127.212,E2 -8127.212} C_VEL
LIN {X 0,Y 577.316,Z 349.306,A -85,B 0,C 180,E1 -8130.4,E2 -8130.4} C_VEL
LIN {X 0,Y 577.266,Z 349.307,A -85,B 0,C 180,E1 -8133.542,E2 -8133.542} C_VEL
LIN {X 0,Y 577.279,Z 349.31,A -85,B 0,C 180,E1 -8136.849,E2 -8136.849} C_VEL
LIN {X 0,Y 577.282,Z 349.311,A -85,B 0,C 180,E1 -8139.888,E2 -8139.888} C_VEL
LIN {X 0,Y 577.263,Z 349.286,A -85,B 0,C 180,E1 -8143.179,E2 -8143.179} C_VEL
LIN {X 0,Y 577.319,Z 349.314,A -85,B 0,C 180,E1 -8146.383,E2 -8146.383} C_VEL
LIN {X 0,Y 577.364,Z 349.61,A -85,B 0,C 180,E1 -8146.522,E2 -8146.522} C_VEL
LIN {X 0,Y 578.083,Z 351.909,A -85,B 0,C 180,E1 -8146.808,E2 -8146.808} C_VEL
LIN {X 0,Y 589.065,Z 368.125,A -85,B 0,C 180,E1 -8148.119,E2 -8148.119} C_VEL
LIN {X 0,Y 599.651,Z 384.804,A -85,B 0,C 180,E1 -8149.331,E2 -8149.331} C_VEL
LIN {X 0,Y 611.538,Z 404.499,A -85,B 0,C 180,E1 -8150.632,E2 -8150.632} C_VEL
LIN {X 0,Y 608.331,Z 552.182,A -85,B 0,C 180,E1 -8152.602,E2 -8152.602} C_VEL
LIN {X 0,Y 607.39,Z 559.879,A -85,B 0,C 180,E1 -8152.645,E2 -8152.645} C_VEL
LIN {X 0,Y 602.071,Z 580.427,A -85,B 0,C 180,E1 -8152.545,E2 -8152.545} C_VEL
LIN {X 0,Y 601.344,Z 587.031,A -85,B 0,C 180,E1 -8152.588,E2 -8152.588} C_VEL
LIN {X 0,Y 597.896,Z 739.693,A -85,B 0,C 180,E1 -8154.636,E2 -8154.636} C_VEL
LIN {X 0,Y 596.657,Z 765.553,A -85,B 0,C 180,E1 -8155.148,E2 -8155.148} C_VEL
LIN {X 0,Y 595.299,Z 786.138,A -85,B 0,C 180,E1 -8155.697,E2 -8155.697} C_VEL
LIN {X 0,Y 593.462,Z 809.785,A -85,B 0,C 180,E1 -8156.491,E2 -8156.491} C_VEL
LIN {X 0,Y 591.452,Z 830.775,A -85,B 0,C 180,E1 -8157.365,E2 -8157.365} C_VEL
LIN {X 0,Y 589.403,Z 850.476,A -85,B 0,C 180,E1 -8158.328,E2 -8158.328} C_VEL
LIN {X 0,Y 586.743,Z 873.279,A -85,B 0,C 180,E1 -8159.65,E2 -8159.65} C_VEL
LIN {X 0,Y 584.411,Z 892.18,A -85,B 0,C 180,E1 -8160.928,E2 -8160.928} C_VEL
LIN {X 0,Y 581.704,Z 913.116,A -85,B 0,C 180,E1 -8162.57,E2 -8162.57} C_VEL
LIN {X 0,Y 579.405,Z 930.214,A -85,B 0,C 180,E1 -8164.112,E2 -8164.112} C_VEL
LIN {X 0,Y 576.902,Z 949.117,A -85,B 0,C 180,E1 -8166.073,E2 -8166.073} C_VEL
LIN {X 0,Y 574.971,Z 963.88,A -85,B 0,C 180,E1 -8167.829,E2 -8167.829} C_VEL
LIN {X 0,Y 573.009,Z 979.861,A -85,B 0,C 180,E1 -8170,E2 -8170} C_VEL
LIN {X 0,Y 571.557,Z 992.364,A -85,B 0,C 180,E1 -8171.962,E2 -8171.962} C_VEL
LIN {X 0,Y 570.304,Z 1004.995,A -85,B 0,C 180,E1 -8174.231,E2 -8174.231} C_VEL
LIN {X 0,Y 569.362,Z 1015.611,A -85,B 0,C 180,E1 -8176.493,E2 -8176.493} C_VEL
LIN {X 0,Y 568.703,Z 1025.057,A -85,B 0,C 180,E1 -8178.849,E2 -8178.849} C_VEL
LIN {X 0,Y 568.28,Z 1032.626,A -85,B 0,C 180,E1 -8181.195,E2 -8181.195} C_VEL
LIN {X 0,Y 568.051,Z 1038.751,A -85,B 0,C 180,E1 -8183.532,E2 -8183.532} C_VEL
LIN {X 0,Y 567.949,Z 1043.461,A -85,B 0,C 180,E1 -8185.962,E2 -8185.962} C_VEL
LIN {X 0,Y 567.919,Z 1046.319,A -85,B 0,C 180,E1 -8188.083,E2 -8188.083} C_VEL
LIN {X 0,Y 567.901,Z 1048.16,A -85,B 0,C 180,E1 -8190.504,E2 -8190.504} C_VEL
LIN {X 0,Y 567.897,Z 1048.354,A -85,B 0,C 180,E1 -8192.725,E2 -8192.725} C_VEL
LIN {X 0,Y 567.9,Z 1047.431,A -85,B 0,C 180,E1 -8194.761,E2 -8194.761} C_VEL
LIN {X 0,Y 567.933,Z 1044.955,A -85,B 0,C 180,E1 -8197.181,E2 -8197.181} C_VEL
LIN {X 0,Y 567.988,Z 1040.906,A -85,B 0,C 180,E1 -8199.525,E2 -8199.525} C_VEL
LIN {X 0,Y 568.157,Z 1035.504,A -85,B 0,C 180,E1 -8201.883,E2 -8201.883} C_VEL
LIN {X 0,Y 568.499,Z 1028.326,A -85,B 0,C 180,E1 -8204.276,E2 -8204.276} C_VEL
LIN {X 0,Y 568.971,Z 1020.772,A -85,B 0,C 180,E1 -8206.357,E2 -8206.357} C_VEL
LIN {X 0,Y 569.837,Z 1010.002,A -85,B 0,C 180,E1 -8208.836,E2 -8208.836} C_VEL
LIN {X 0,Y 570.781,Z 999.79,A -85,B 0,C 180,E1 -8210.831,E2 -8210.831} C_VEL
LIN {X 0,Y 572.206,Z 986.821,A -85,B 0,C 180,E1 -8213.043,E2 -8213.043} C_VEL
LIN {X 0,Y 573.828,Z 973.072,A -85,B 0,C 180,E1 -8215.051,E2 -8215.051} C_VEL
LIN {X 0,Y 575.83,Z 957.495,A -85,B 0,C 180,E1 -8217.061,E2 -8217.061} C_VEL
LIN {X 0,Y 578.075,Z 940.311,A -85,B 0,C 180,E1 -8218.967,E2 -8218.967} C_VEL
LIN {X 0,Y 580.412,Z 923.055,A -85,B 0,C 180,E1 -8220.659,E2 -8220.659} C_VEL
LIN {X 0,Y 582.952,Z 903.733,A -85,B 0,C 180,E1 -8222.296,E2 -8222.296} C_VEL
LIN {X 0,Y 585.365,Z 885.323,A -85,B 0,C 180,E1 -8223.662,E2 -8223.662} C_VEL
LIN {X 0,Y 588.092,Z 863.106,A -85,B 0,C 180,E1 -8225.077,E2 -8225.077} C_VEL
LIN {X 0,Y 590.248,Z 843.978,A -85,B 0,C 180,E1 -8226.123,E2 -8226.123} C_VEL
LIN {X 0,Y 592.648,Z 820.801,A -85,B 0,C 180,E1 -8227.194,E2 -8227.194} C_VEL
LIN {X 0,Y 594.487,Z 799.765,A -85,B 0,C 180,E1 -8227.995,E2 -8227.995} C_VEL
LIN {X 0,Y 596.337,Z 775.952,A -85,B 0,C 180,E1 -8228.729,E2 -8228.729} C_VEL
LIN {X 0,Y 597.667,Z 752.905,A -85,B 0,C 180,E1 -8229.258,E2 -8229.258} C_VEL
LIN {X 0,Y 598.602,Z 729.735,A -85,B 0,C 180,E1 -8229.649,E2 -8229.649} C_VEL
LIN {X 0,Y 604.506,Z 476.957,A -85,B 0,C 180,E1 -8233.049,E2 -8233.049} C_VEL
LIN {X 0,Y 606.086,Z 407.629,A -85,B 0,C 180,E1 -8234.004,E2 -8234.004} C_VEL
LIN {X 0,Y 594.518,Z 388.483,A -85,B 0,C 180,E1 -8235.364,E2 -8235.364} C_VEL
LIN {X 0,Y 581.143,Z 368.229,A -85,B 0,C 180,E1 -8237.017,E2 -8237.017} C_VEL
LIN {X 0,Y 571.846,Z 355.177,A -85,B 0,C 180,E1 -8238.226,E2 -8238.226} C_VEL
LIN {X 0,Y 569.806,Z 352.204,A -85,B 0,C 180,E1 -8238.502,E2 -8238.502} C_VEL
LIN {X 0,Y 569.318,Z 350.274,A -85,B 0,C 180,E1 -8238.806,E2 -8238.806} C_VEL
LIN {X 0,Y 569.353,Z 350.309,A -85,B 0,C 180,E1 -8242.072,E2 -8242.072} C_VEL
LIN {X 0,Y 569.337,Z 350.272,A -85,B 0,C 180,E1 -8245.195,E2 -8245.195} C_VEL
LIN {X 0,Y 569.33,Z 350.299,A -85,B 0,C 180,E1 -8248.442,E2 -8248.442} C_VEL
LIN {X 0,Y 569.355,Z 350.299,A -85,B 0,C 180,E1 -8251.466,E2 -8251.466} C_VEL
LIN {X 0,Y 569.32,Z 350.299,A -85,B 0,C 180,E1 -8254.754,E2 -8254.754} C_VEL
LIN {X 0,Y 569.39,Z 350.293,A -85,B 0,C 180,E1 -8257.926,E2 -8257.926} C_VEL
LIN {X 0,Y 569.322,Z 350.31,A -85,B 0,C 180,E1 -8261.146,E2 -8261.146} C_VEL
LIN {X 0,Y 569.353,Z 350.307,A -85,B 0,C 180,E1 -8264.413,E2 -8264.413} C_VEL
LIN {X 0,Y 569.328,Z 350.307,A -85,B 0,C 180,E1 -8267.421,E2 -8267.421} C_VEL
LIN {X 0,Y 569.329,Z 350.303,A -85,B 0,C 180,E1 -8270.804,E2 -8270.804} C_VEL
LIN {X 0,Y 569.354,Z 350.297,A -85,B 0,C 180,E1 -8273.85,E2 -8273.85} C_VEL
LIN {X 0,Y 569.32,Z 350.309,A -85,B 0,C 180,E1 -8277.081,E2 -8277.081} C_VEL
LIN {X 0,Y 569.39,Z 350.306,A -85,B 0,C 180,E1 -8280.302,E2 -8280.302} C_VEL
LIN {X 0,Y 569.318,Z 350.298,A -85,B 0,C 180,E1 -8283.524,E2 -8283.524} C_VEL
LIN {X 0,Y 569.354,Z 350.291,A -85,B 0,C 180,E1 -8286.757,E2 -8286.757} C_VEL
LIN {X 0,Y 569.33,Z 350.313,A -85,B 0,C 180,E1 -8289.85,E2 -8289.85} C_VEL
LIN {X 0,Y 569.327,Z 350.309,A -85,B 0,C 180,E1 -8293.198,E2 -8293.198} C_VEL
LIN {X 0,Y 569.35,Z 350.295,A -85,B 0,C 180,E1 -8296.215,E2 -8296.215} C_VEL
LIN {X 0,Y 569.316,Z 350.293,A -85,B 0,C 180,E1 -8299.493,E2 -8299.493} C_VEL
LIN {X 0,Y 569.39,Z 350.292,A -85,B 0,C 180,E1 -8302.618,E2 -8302.618} C_VEL
LIN {X 0,Y 569.318,Z 350.312,A -85,B 0,C 180,E1 -8305.821,E2 -8305.821} C_VEL
LIN {X 0,Y 569.361,Z 350.307,A -85,B 0,C 180,E1 -8309.108,E2 -8309.108} C_VEL
LIN {X 0,Y 569.326,Z 350.313,A -85,B 0,C 180,E1 -8312.165,E2 -8312.165} C_VEL
LIN {X 0,Y 569.326,Z 350.314,A -85,B 0,C 180,E1 -8315.595,E2 -8315.595} C_VEL
LIN {X 0,Y 569.372,Z 350.309,A -85,B 0,C 180,E1 -8318.765,E2 -8318.765} C_VEL
LIN {X 0,Y 569.391,Z 350.343,A -85,B 0,C 180,E1 -8321.054,E2 -8321.054} C_VEL
LIN {X 0,Y 570.724,Z 353.923,A -85,B 0,C 180,E1 -8321.606,E2 -8321.606} C_VEL
LIN {X 0,Y 576.48,Z 367.303,A -85,B 0,C 180,E1 -8323.674,E2 -8323.674} C_VEL
LIN {X 0,Y 579.172,Z 373.346,A -85,B 0,C 180,E1 -8324.536,E2 -8324.536} C_VEL
LIN {X 0,Y 591.403,Z 392.552,A -85,B 0,C 180,E1 -8326.075,E2 -8326.075} C_VEL
LIN {X 0,Y 603.345,Z 412.578,A -85,B 0,C 180,E1 -8327.499,E2 -8327.499} C_VEL
LIN {X 0,Y 605.431,Z 416.842,A -85,B 0,C 180,E1 -8327.751,E2 -8327.751} C_VEL
LIN {X 0,Y 606.136,Z 421.288,A -85,B 0,C 180,E1 -8327.883,E2 -8327.883} C_VEL
LIN {X 0,Y 599.948,Z 683.573,A -85,B 0,C 180,E1 -8331.422,E2 -8331.422} C_VEL
LIN {X 0,Y 597.954,Z 766.151,A -85,B 0,C 180,E1 -8332.546,E2 -8332.546} C_VEL
LIN {X 0,Y 596.563,Z 791.68,A -85,B 0,C 180,E1 -8333.052,E2 -8333.052} C_VEL
LIN {X 0,Y 595.033,Z 813.35,A -85,B 0,C 180,E1 -8333.632,E2 -8333.632} C_VEL
LIN {X 0,Y 592.944,Z 838.191,A -85,B 0,C 180,E1 -8334.484,E2 -8334.484} C_VEL
LIN {X 0,Y 591.005,Z 857.874,A -85,B 0,C 180,E1 -8335.31,E2 -8335.31} C_VEL
LIN {X 0,Y 588.696,Z 879.583,A -85,B 0,C 180,E1 -8336.378,E2 -8336.378} C_VEL
LIN {X 0,Y 586.075,Z 901.435,A -85,B 0,C 180,E1 -8337.666,E2 -8337.666} C_VEL
LIN {X 0,Y 583.562,Z 922.052,A -85,B 0,C 180,E1 -8339.068,E2 -8339.068} C_VEL
LIN {X 0,Y 581.016,Z 941.713,A -85,B 0,C 180,E1 -8340.629,E2 -8340.629} C_VEL
LIN {X 0,Y 578.769,Z 959.142,A -85,B 0,C 180,E1 -8342.195,E2 -8342.195} C_VEL
LIN {X 0,Y 576.447,Z 977.418,A -85,B 0,C 180,E1 -8344.08,E2 -8344.08} C_VEL
LIN {X 0,Y 574.577,Z 992.602,A -85,B 0,C 180,E1 -8345.861,E2 -8345.861} C_VEL
LIN {X 0,Y 572.69,Z 1008.981,A -85,B 0,C 180,E1 -8348.06,E2 -8348.06} C_VEL
LIN {X 0,Y 571.321,Z 1021.701,A -85,B 0,C 180,E1 -8350.023,E2 -8350.023} C_VEL
LIN {X 0,Y 570.111,Z 1034.747,A -85,B 0,C 180,E1 -8352.337,E2 -8352.337} C_VEL
LIN {X 0,Y 569.304,Z 1044.734,A -85,B 0,C 180,E1 -8354.412,E2 -8354.412} C_VEL
LIN {X 0,Y 568.673,Z 1054.558,A -85,B 0,C 180,E1 -8356.787,E2 -8356.787} C_VEL
LIN {X 0,Y 568.282,Z 1062.131,A -85,B 0,C 180,E1 -8359.053,E2 -8359.053} C_VEL
LIN {X 0,Y 568.057,Z 1067.991,A -85,B 0,C 180,E1 -8361.191,E2 -8361.191} C_VEL
LIN {X 0,Y 567.95,Z 1073.173,A -85,B 0,C 180,E1 -8363.734,E2 -8363.734} C_VEL
LIN {X 0,Y 567.913,Z 1076.121,A -85,B 0,C 180,E1 -8365.86,E2 -8365.86} C_VEL
LIN {X 0,Y 567.903,Z 1077.97,A -85,B 0,C 180,E1 -8368.083,E2 -8368.083} C_VEL
LIN {X 0,Y 567.895,Z 1078.393,A -85,B 0,C 180,E1 -8370.504,E2 -8370.504} C_VEL
LIN {X 0,Y 567.907,Z 1077.493,A -85,B 0,C 180,E1 -8372.624,E2 -8372.624} C_VEL
LIN {X 0,Y 567.93,Z 1075.21,A -85,B 0,C 180,E1 -8374.949,E2 -8374.949} C_VEL
LIN {X 0,Y 567.987,Z 1071.101,A -85,B 0,C 180,E1 -8377.383,E2 -8377.383} C_VEL
LIN {X 0,Y 568.109,Z 1066.7,A -85,B 0,C 180,E1 -8379.319,E2 -8379.319} C_VEL
LIN {X 0,Y 568.39,Z 1059.935,A -85,B 0,C 180,E1 -8381.672,E2 -8381.672} C_VEL
LIN {X 0,Y 568.853,Z 1051.423,A -85,B 0,C 180,E1 -8384.006,E2 -8384.006} C_VEL
LIN {X 0,Y 569.527,Z 1041.953,A -85,B 0,C 180,E1 -8386.209,E2 -8386.209} C_VEL
LIN {X 0,Y 570.518,Z 1030.094,A -85,B 0,C 180,E1 -8388.529,E2 -8388.529} C_VEL
LIN {X 0,Y 571.654,Z 1018.64,A -85,B 0,C 180,E1 -8390.477,E2 -8390.477} C_VEL
LIN {X 0,Y 573.357,Z 1003.045,A -85,B 0,C 180,E1 -8392.777,E2 -8392.777} C_VEL
LIN {X 0,Y 575.004,Z 989.123,A -85,B 0,C 180,E1 -8394.569,E2 -8394.569} C_VEL
LIN {X 0,Y 577.244,Z 971.16,A -85,B 0,C 180,E1 -8396.601,E2 -8396.601} C_VEL
LIN {X 0,Y 579.352,Z 954.7,A -85,B 0,C 180,E1 -8398.222,E2 -8398.222} C_VEL
LIN {X 0,Y 581.832,Z 935.519,A -85,B 0,C 180,E1 -8399.892,E2 -8399.892} C_VEL
LIN {X 0,Y 584.245,Z 916.026,A -85,B 0,C 180,E1 -8401.35,E2 -8401.35} C_VEL
LIN {X 0,Y 586.781,Z 895.477,A -85,B 0,C 180,E1 -8402.696,E2 -8402.696} C_VEL
LIN {X 0,Y 589.214,Z 873.399,A -85,B 0,C 180,E1 -8403.919,E2 -8403.919} C_VEL
LIN {X 0,Y 591.294,Z 853.527,A -85,B 0,C 180,E1 -8404.859,E2 -8404.859} C_VEL
LIN {X 0,Y 593.524,Z 828.734,A -85,B 0,C 180,E1 -8405.833,E2 -8405.833} C_VEL
LIN {X 0,Y 595.213,Z 807.274,A -85,B 0,C 180,E1 -8406.508,E2 -8406.508} C_VEL
LIN {X 0,Y 596.905,Z 781.183,A -85,B 0,C 180,E1 -8407.135,E2 -8407.135} C_VEL
LIN {X 0,Y 597.85,Z 759.335,A -85,B 0,C 180,E1 -8407.513,E2 -8407.513} C_VEL
LIN {X 0,Y 603.083,Z 519.98,A -85,B 0,C 180,E1 -8410.708,E2 -8410.708} C_VEL
LIN {X 0,Y 605.254,Z 419.539,A -85,B 0,C 180,E1 -8412.07,E2 -8412.07} C_VEL
LIN {X 0,Y 604.046,Z 415.086,A -85,B 0,C 180,E1 -8412.239,E2 -8412.239} C_VEL
LIN {X 0,Y 589.277,Z 390.002,A -85,B 0,C 180,E1 -8413.921,E2 -8413.921} C_VEL
LIN {X 0,Y 578.551,Z 372.701,A -85,B 0,C 180,E1 -8415.236,E2 -8415.236} C_VEL
LIN {X 0,Y 572.143,Z 357.34,A -85,B 0,C 180,E1 -8417.442,E2 -8417.442} C_VEL
LIN {X 0,Y 569.373,Z 350.571,A -85,B 0,C 180,E1 -8418.453,E2 -8418.453} C_VEL
LIN {X 0,Y 569.371,Z 350.305,A -85,B 0,C 180,E1 -8419.21,E2 -8419.21} C_VEL
LIN {X 0,Y 569.319,Z 350.305,A -85,B 0,C 180,E1 -8422.216,E2 -8422.216} C_VEL
LIN {X 0,Y 569.353,Z 350.297,A -85,B 0,C 180,E1 -8425.452,E2 -8425.452} C_VEL
LIN {X 0,Y 569.322,Z 350.302,A -85,B 0,C 180,E1 -8428.441,E2 -8428.441} C_VEL
LIN {X 0,Y 569.331,Z 350.299,A -85,B 0,C 180,E1 -8431.841,E2 -8431.841} C_VEL
LIN {X 0,Y 569.361,Z 350.307,A -85,B 0,C 180,E1 -8434.982,E2 -8434.982} C_VEL
LIN {X 0,Y 569.319,Z 350.312,A -85,B 0,C 180,E1 -8438.14,E2 -8438.14} C_VEL
LIN {X 0,Y 569.373,Z 350.288,A -85,B 0,C 180,E1 -8441.254,E2 -8441.254} C_VEL
LIN {X 0,Y 569.317,Z 350.305,A -85,B 0,C 180,E1 -8444.412,E2 -8444.412} C_VEL
LIN {X 0,Y 569.381,Z 350.303,A -85,B 0,C 180,E1 -8447.526,E2 -8447.526} C_VEL
LIN {X 0,Y 569.318,Z 350.289,A -85,B 0,C 180,E1 -8450.701,E2 -8450.701} C_VEL
LIN {X 0,Y 569.354,Z 350.303,A -85,B 0,C 180,E1 -8453.951,E2 -8453.951} C_VEL
LIN {X 0,Y 569.335,Z 350.302,A -85,B 0,C 180,E1 -8457.081,E2 -8457.081} C_VEL
LIN {X 0,Y 569.324,Z 350.288,A -85,B 0,C 180,E1 -8460.403,E2 -8460.403} C_VEL
LIN {X 0,Y 569.366,Z 350.307,A -85,B 0,C 180,E1 -8463.524,E2 -8463.524} C_VEL
LIN {X 0,Y 569.317,Z 350.298,A -85,B 0,C 180,E1 -8466.758,E2 -8466.758} C_VEL
LIN {X 0,Y 569.378,Z 350.295,A -85,B 0,C 180,E1 -8469.91,E2 -8469.91} C_VEL
LIN {X 0,Y 569.323,Z 350.309,A -85,B 0,C 180,E1 -8473.095,E2 -8473.095} C_VEL
LIN {X 0,Y 569.355,Z 350.29,A -85,B 0,C 180,E1 -8476.319,E2 -8476.319} C_VEL
LIN {X 0,Y 569.335,Z 350.308,A -85,B 0,C 180,E1 -8479.421,E2 -8479.421} C_VEL
LIN {X 0,Y 569.33,Z 350.313,A -85,B 0,C 180,E1 -8482.775,E2 -8482.775} C_VEL
LIN {X 0,Y 569.372,Z 350.288,A -85,B 0,C 180,E1 -8485.955,E2 -8485.955} C_VEL
LIN {X 0,Y 569.321,Z 350.295,A -85,B 0,C 180,E1 -8489.11,E2 -8489.11} C_VEL
LIN {X 0,Y 569.385,Z 350.3,A -85,B 0,C 180,E1 -8492.266,E2 -8492.266} C_VEL
LIN {X 0,Y 569.325,Z 350.311,A -85,B 0,C 180,E1 -8495.422,E2 -8495.422} C_VEL
LIN {X 0,Y 569.36,Z 350.309,A -85,B 0,C 180,E1 -8498.697,E2 -8498.697} C_VEL
LIN {X 0,Y 569.333,Z 350.316,A -85,B 0,C 180,E1 -8501.73,E2 -8501.73} C_VEL
LIN {X 0,Y 569.331,Z 350.266,A -85,B 0,C 180,E1 -8505.089,E2 -8505.089} C_VEL
LIN {X 0,Y 569.339,Z 350.369,A -85,B 0,C 180,E1 -8505.77,E2 -8505.77} C_VEL
LIN {X 0,Y 569.864,Z 352.293,A -85,B 0,C 180,E1 -8505.993,E2 -8505.993} C_VEL
LIN {X 0,Y 571.953,Z 355.251,A -85,B 0,C 180,E1 -8506.257,E2 -8506.257} C_VEL
LIN {X 0,Y 584.357,Z 373.532,A -85,B 0,C 180,E1 -8507.772,E2 -8507.772} C_VEL
LIN {X 0,Y 595.034,Z 390.48,A -85,B 0,C 180,E1 -8509.018,E2 -8509.018} C_VEL
LIN {X 0,Y 605.418,Z 407.827,A -85,B 0,C 180,E1 -8510.18,E2 -8510.18} C_VEL
LIN {X 0,Y 601.344,Z 587.031,A -85,B 0,C 180,E1 -8512.588,E2 -8512.588} C_VEL
LIN {X 0,Y 600.399,Z 594.727,A -85,B 0,C 180,E1 -8512.631,E2 -8512.631} C_VEL
LIN {X 0,Y 595.054,Z 615.267,A -85,B 0,C 180,E1 -8512.528,E2 -8512.528} C_VEL
LIN {X 0,Y 594.323,Z 621.871,A -85,B 0,C 180,E1 -8512.571,E2 -8512.571} C_VEL
LIN {X 0,Y 591.491,Z 740.275,A -85,B 0,C 180,E1 -8514.178,E2 -8514.178} C_VEL
LIN {X 0,Y 590.199,Z 765.933,A -85,B 0,C 180,E1 -8514.692,E2 -8514.692} C_VEL
LIN {X 0,Y 588.778,Z 786.603,A -85,B 0,C 180,E1 -8515.248,E2 -8515.248} C_VEL
LIN {X 0,Y 586.911,Z 809.672,A -85,B 0,C 180,E1 -8516.027,E2 -8516.027} C_VEL
LIN {X 0,Y 584.739,Z 831.447,A -85,B 0,C 180,E1 -8516.942,E2 -8516.942} C_VEL
LIN {X 0,Y 582.598,Z 851.106,A -85,B 0,C 180,E1 -8517.915,E2 -8517.915} C_VEL
LIN {X 0,Y 579.921,Z 873.043,A -85,B 0,C 180,E1 -8519.197,E2 -8519.197} C_VEL
LIN {X 0,Y 577.554,Z 891.278,A -85,B 0,C 180,E1 -8520.435,E2 -8520.435} C_VEL
LIN {X 0,Y 574.708,Z 912.427,A -85,B 0,C 180,E1 -8522.095,E2 -8522.095} C_VEL
LIN {X 0,Y 572.362,Z 929.084,A -85,B 0,C 180,E1 -8523.602,E2 -8523.602} C_VEL
LIN {X 0,Y 569.881,Z 946.877,A -85,B 0,C 180,E1 -8525.428,E2 -8525.428} C_VEL
LIN {X 0,Y 567.593,Z 963.267,A -85,B 0,C 180,E1 -8527.384,E2 -8527.384} C_VEL
LIN {X 0,Y 565.641,Z 978.22,A -85,B 0,C 180,E1 -8529.404,E2 -8529.404} C_VEL
LIN {X 0,Y 563.908,Z 992.141,A -85,B 0,C 180,E1 -8531.602,E2 -8531.602} C_VEL
LIN {X 0,Y 562.601,Z 1004.328,A -85,B 0,C 180,E1 -8533.798,E2 -8533.798} C_VEL
LIN {X 0,Y 561.55,Z 1015.061,A -85,B 0,C 180,E1 -8536.091,E2 -8536.091} C_VEL
LIN {X 0,Y 560.865,Z 1023.83,A -85,B 0,C 180,E1 -8538.274,E2 -8538.274} C_VEL
LIN {X 0,Y 560.352,Z 1032.037,A -85,B 0,C 180,E1 -8540.759,E2 -8540.759} C_VEL
LIN {X 0,Y 560.1,Z 1037.791,A -85,B 0,C 180,E1 -8542.924,E2 -8542.924} C_VEL
LIN {X 0,Y 559.965,Z 1042.874,A -85,B 0,C 180,E1 -8545.391,E2 -8545.391} C_VEL
LIN {X 0,Y 559.925,Z 1046.117,A -85,B 0,C 180,E1 -8547.748,E2 -8547.748} C_VEL
LIN {X 0,Y 559.918,Z 1047.976,A -85,B 0,C 180,E1 -8550,E2 -8550} C_VEL
LIN {X 0,Y 559.896,Z 1048.458,A -85,B 0,C 180,E1 -8552.559,E2 -8552.559} C_VEL
LIN {X 0,Y 559.901,Z 1047.57,A -85,B 0,C 180,E1 -8554.712,E2 -8554.712} C_VEL
LIN {X 0,Y 559.937,Z 1045.192,A -85,B 0,C 180,E1 -8557.181,E2 -8557.181} C_VEL
LIN {X 0,Y 559.998,Z 1041.245,A -85,B 0,C 180,E1 -8559.558,E2 -8559.558} C_VEL
LIN {X 0,Y 560.165,Z 1036.402,A -85,B 0,C 180,E1 -8561.741,E2 -8561.741} C_VEL
LIN {X 0,Y 560.544,Z 1028.866,A -85,B 0,C 180,E1 -8564.356,E2 -8564.356} C_VEL
LIN {X 0,Y 561.057,Z 1021.218,A -85,B 0,C 180,E1 -8566.503,E2 -8566.503} C_VEL
LIN {X 0,Y 561.93,Z 1011.097,A -85,B 0,C 180,E1 -8568.896,E2 -8568.896} C_VEL
LIN {X 0,Y 562.978,Z 1000.415,A -85,B 0,C 180,E1 -8571.024,E2 -8571.024} C_VEL
LIN {X 0,Y 564.484,Z 987.53,A -85,B 0,C 180,E1 -8573.266,E2 -8573.266} C_VEL
LIN {X 0,Y 566.302,Z 973.067,A -85,B 0,C 180,E1 -8575.407,E2 -8575.407} C_VEL
LIN {X 0,Y 568.423,Z 957.461,A -85,B 0,C 180,E1 -8577.443,E2 -8577.443} C_VEL
LIN {X 0,Y 570.744,Z 940.758,A -85,B 0,C 180,E1 -8579.318,E2 -8579.318} C_VEL
LIN {X 0,Y 573.203,Z 923.555,A -85,B 0,C 180,E1 -8581.029,E2 -8581.029} C_VEL
LIN {X 0,Y 575.887,Z 904.313,A -85,B 0,C 180,E1 -8582.682,E2 -8582.682} C_VEL
LIN {X 0,Y 578.42,Z 885.955,A -85,B 0,C 180,E1 -8584.062,E2 -8584.062} C_VEL
LIN {X 0,Y 581.277,Z 863.847,A -85,B 0,C 180,E1 -8585.49,E2 -8585.49} C_VEL
LIN {X 0,Y 583.53,Z 844.808,A -85,B 0,C 180,E1 -8586.543,E2 -8586.543} C_VEL
LIN {X 0,Y 585.978,Z 822.583,A -85,B 0,C 180,E1 -8587.591,E2 -8587.591} C_VEL
LIN {X 0,Y 588.031,Z 800.135,A -85,B 0,C 180,E1 -8588.457,E2 -8588.457} C_VEL
LIN {X 0,Y 589.972,Z 776.277,A -85,B 0,C 180,E1 -8589.198,E2 -8589.198} C_VEL
LIN {X 0,Y 591.359,Z 753.251,A -85,B 0,C 180,E1 -8589.731,E2 -8589.731} C_VEL
LIN {X 0,Y 592.323,Z 730.378,A -85,B 0,C 180,E1 -8590.122,E2 -8590.122} C_VEL
LIN {X 0,Y 598.539,Z 477.791,A -85,B 0,C 180,E1 -8593.551,E2 -8593.551} C_VEL
LIN {X 0,Y 600.073,Z 410.838,A -85,B 0,C 180,E1 -8594.488,E2 -8594.488} C_VEL
LIN {X 0,Y 587.214,Z 389.608,A -85,B 0,C 180,E1 -8596.045,E2 -8596.045} C_VEL
LIN {X 0,Y 573.32,Z 368.918,A -85,B 0,C 180,E1 -8597.82,E2 -8597.82} C_VEL
LIN {X 0,Y 567.731,Z 361.268,A -85,B 0,C 180,E1 -8598.565,E2 -8598.565} C_VEL
LIN {X 0,Y 564.464,Z 356.623,A -85,B 0,C 180,E1 -8599.015,E2 -8599.015} C_VEL
LIN {X 0,Y 562.218,Z 353.874,A -85,B 0,C 180,E1 -8599.321,E2 -8599.321} C_VEL
LIN {X 0,Y 561.563,Z 351.979,A -85,B 0,C 180,E1 -8599.466,E2 -8599.466} C_VEL
LIN {X 0,Y 561.445,Z 351.25,A -85,B 0,C 180,E1 -8599.589,E2 -8599.589} C_VEL
LIN {X 0,Y 561.381,Z 351.276,A -85,B 0,C 180,E1 -8602.765,E2 -8602.765} C_VEL
LIN {X 0,Y 561.417,Z 351.281,A -85,B 0,C 180,E1 -8606.094,E2 -8606.094} C_VEL
LIN {X 0,Y 561.401,Z 351.292,A -85,B 0,C 180,E1 -8609.258,E2 -8609.258} C_VEL
LIN {X 0,Y 561.387,Z 351.299,A -85,B 0,C 180,E1 -8612.643,E2 -8612.643} C_VEL
LIN {X 0,Y 561.441,Z 351.289,A -85,B 0,C 180,E1 -8615.819,E2 -8615.819} C_VEL
LIN {X 0,Y 561.381,Z 351.291,A -85,B 0,C 180,E1 -8619.022,E2 -8619.022} C_VEL
LIN {X 0,Y 561.424,Z 351.283,A -85,B 0,C 180,E1 -8622.269,E2 -8622.269} C_VEL
LIN {X 0,Y 561.386,Z 351.293,A -85,B 0,C 180,E1 -8625.35,E2 -8625.35} C_VEL
LIN {X 0,Y 561.389,Z 351.296,A -85,B 0,C 180,E1 -8628.805,E2 -8628.805} C_VEL
LIN {X 0,Y 561.437,Z 351.298,A -85,B 0,C 180,E1 -8632.015,E2 -8632.015} C_VEL
LIN {X 0,Y 561.379,Z 351.292,A -85,B 0,C 180,E1 -8635.198,E2 -8635.198} C_VEL
LIN {X 0,Y 561.433,Z 351.279,A -85,B 0,C 180,E1 -8638.469,E2 -8638.469} C_VEL
LIN {X 0,Y 561.384,Z 351.301,A -85,B 0,C 180,E1 -8641.531,E2 -8641.531} C_VEL
LIN {X 0,Y 561.4,Z 351.299,A -85,B 0,C 180,E1 -8644.904,E2 -8644.904} C_VEL
LIN {X 0,Y 561.401,Z 351.285,A -85,B 0,C 180,E1 -8647.986,E2 -8647.986} C_VEL
LIN {X 0,Y 561.38,Z 351.281,A -85,B 0,C 180,E1 -8651.299,E2 -8651.299} C_VEL
LIN {X 0,Y 561.448,Z 351.281,A -85,B 0,C 180,E1 -8654.543,E2 -8654.543} C_VEL
LIN {X 0,Y 561.382,Z 351.3,A -85,B 0,C 180,E1 -8657.733,E2 -8657.733} C_VEL
LIN {X 0,Y 561.412,Z 351.298,A -85,B 0,C 180,E1 -8661.052,E2 -8661.052} C_VEL
LIN {X 0,Y 561.388,Z 351.287,A -85,B 0,C 180,E1 -8664.071,E2 -8664.071} C_VEL
LIN {X 0,Y 561.386,Z 351.288,A -85,B 0,C 180,E1 -8667.502,E2 -8667.502} C_VEL
LIN {X 0,Y 561.419,Z 351.3,A -85,B 0,C 180,E1 -8670.503,E2 -8670.503} C_VEL
LIN {X 0,Y 561.38,Z 351.303,A -85,B 0,C 180,E1 -8673.76,E2 -8673.76} C_VEL
LIN {X 0,Y 561.441,Z 351.299,A -85,B 0,C 180,E1 -8677.01,E2 -8677.01} C_VEL
LIN {X 0,Y 561.382,Z 351.304,A -85,B 0,C 180,E1 -8680.173,E2 -8680.173} C_VEL
LIN {X 0,Y 561.555,Z 352.203,A -85,B 0,C 180,E1 -8680.352,E2 -8680.352} C_VEL
LIN {X 0,Y 563.435,Z 356.303,A -85,B 0,C 180,E1 -8681.043,E2 -8681.043} C_VEL
LIN {X 0,Y 569.718,Z 370.71,A -85,B 0,C 180,E1 -8683.333,E2 -8683.333} C_VEL
LIN {X 0,Y 570.766,Z 373.125,A -85,B 0,C 180,E1 -8683.648,E2 -8683.648} C_VEL
LIN {X 0,Y 582.747,Z 391.401,A -85,B 0,C 180,E1 -8685.211,E2 -8685.211} C_VEL
LIN {X 0,Y 595.371,Z 412.407,A -85,B 0,C 180,E1 -8686.775,E2 -8686.775} C_VEL
LIN {X 0,Y 600.003,Z 420.961,A -85,B 0,C 180,E1 -8687.336,E2 -8687.336} C_VEL
LIN {X 0,Y 600.16,Z 425.019,A -85,B 0,C 180,E1 -8687.415,E2 -8687.415} C_VEL
LIN {X 0,Y 593.701,Z 685.414,A -85,B 0,C 180,E1 -8690.959,E2 -8690.959} C_VEL
LIN {X 0,Y 591.65,Z 766.034,A -85,B 0,C 180,E1 -8692.067,E2 -8692.067} C_VEL
LIN {X 0,Y 590.187,Z 791.581,A -85,B 0,C 180,E1 -8692.578,E2 -8692.578} C_VEL
LIN {X 0,Y 588.579,Z 813.335,A -85,B 0,C 180,E1 -8693.164,E2 -8693.164} C_VEL
LIN {X 0,Y 586.38,Z 838.196,A -85,B 0,C 180,E1 -8694.025,E2 -8694.025} C_VEL
LIN {X 0,Y 584.287,Z 858.471,A -85,B 0,C 180,E1 -8694.886,E2 -8694.886} C_VEL
LIN {X 0,Y 581.811,Z 880.444,A -85,B 0,C 180,E1 -8695.986,E2 -8695.986} C_VEL
LIN {X 0,Y 579.215,Z 901.047,A -85,B 0,C 180,E1 -8697.215,E2 -8697.215} C_VEL
LIN {X 0,Y 576.615,Z 921.114,A -85,B 0,C 180,E1 -8698.589,E2 -8698.589} C_VEL
LIN {X 0,Y 573.894,Z 941.134,A -85,B 0,C 180,E1 -8700.188,E2 -8700.188} C_VEL
LIN {X 0,Y 571.553,Z 958.312,A -85,B 0,C 180,E1 -8701.748,E2 -8701.748} C_VEL
LIN {X 0,Y 568.994,Z 977.194,A -85,B 0,C 180,E1 -8703.715,E2 -8703.715} C_VEL
LIN {X 0,Y 567.016,Z 992.376,A -85,B 0,C 180,E1 -8705.518,E2 -8705.518} C_VEL
LIN {X 0,Y 564.997,Z 1008.815,A -85,B 0,C 180,E1 -8707.755,E2 -8707.755} C_VEL
LIN {X 0,Y 563.613,Z 1020.97,A -85,B 0,C 180,E1 -8709.652,E2 -8709.652} C_VEL
LIN {X 0,Y 562.316,Z 1034.002,A -85,B 0,C 180,E1 -8711.977,E2 -8711.977} C_VEL
LIN {X 0,Y 561.398,Z 1044.512,A -85,B 0,C 180,E1 -8714.187,E2 -8714.187} C_VEL
LIN {X 0,Y 560.745,Z 1053.948,A -85,B 0,C 180,E1 -8716.491,E2 -8716.491} C_VEL
LIN {X 0,Y 560.304,Z 1061.89,A -85,B 0,C 180,E1 -8718.888,E2 -8718.888} C_VEL
LIN {X 0,Y 560.065,Z 1067.774,A -85,B 0,C 180,E1 -8721.065,E2 -8721.065} C_VEL
LIN {X 0,Y 559.949,Z 1073.035,A -85,B 0,C 180,E1 -8723.644,E2 -8723.644} C_VEL
LIN {X 0,Y 559.914,Z 1076.033,A -85,B 0,C 180,E1 -8725.801,E2 -8725.801} C_VEL
LIN {X 0,Y 559.904,Z 1077.913,A -85,B 0,C 180,E1 -8728.056,E2 -8728.056} C_VEL
LIN {X 0,Y 559.896,Z 1078.345,A -85,B 0,C 180,E1 -8730.512,E2 -8730.512} C_VEL
LIN {X 0,Y 559.907,Z 1077.429,A -85,B 0,C 180,E1 -8732.661,E2 -8732.661} C_VEL
LIN {X 0,Y 559.931,Z 1075.107,A -85,B 0,C 180,E1 -8735.02,E2 -8735.02} C_VEL
LIN {X 0,Y 559.984,Z 1070.929,A -85,B 0,C 180,E1 -8737.49,E2 -8737.49} C_VEL
LIN {X 0,Y 560.134,Z 1066.227,A -85,B 0,C 180,E1 -8739.556,E2 -8739.556} C_VEL
LIN {X 0,Y 560.464,Z 1058.71,A -85,B 0,C 180,E1 -8742.134,E2 -8742.134} C_VEL
LIN {X 0,Y 560.952,Z 1050.667,A -85,B 0,C 180,E1 -8744.345,E2 -8744.345} C_VEL
LIN {X 0,Y 561.76,Z 1040.359,A -85,B 0,C 180,E1 -8746.743,E2 -8746.743} C_VEL
LIN {X 0,Y 562.796,Z 1028.901,A -85,B 0,C 180,E1 -8748.973,E2 -8748.973} C_VEL
LIN {X 0,Y 564.22,Z 1015.654,A -85,B 0,C 180,E1 -8751.225,E2 -8751.225} C_VEL
LIN {X 0,Y 565.906,Z 1001.267,A -85,B 0,C 180,E1 -8753.315,E2 -8753.315} C_VEL
LIN {X 0,Y 567.913,Z 985.575,A -85,B 0,C 180,E1 -8755.33,E2 -8755.33} C_VEL
LIN {X 0,Y 570.192,Z 968.342,A -85,B 0,C 180,E1 -8757.242,E2 -8757.242} C_VEL
LIN {X 0,Y 572.443,Z 951.643,A -85,B 0,C 180,E1 -8758.879,E2 -8758.879} C_VEL
LIN {X 0,Y 575.208,Z 931.042,A -85,B 0,C 180,E1 -8760.631,E2 -8760.631} C_VEL
LIN {X 0,Y 577.627,Z 912.745,A -85,B 0,C 180,E1 -8761.985,E2 -8761.985} C_VEL
LIN {X 0,Y 580.49,Z 889.767,A -85,B 0,C 180,E1 -8763.449,E2 -8763.449} C_VEL
LIN {X 0,Y 582.689,Z 870.64,A -85,B 0,C 180,E1 -8764.491,E2 -8764.491} C_VEL
LIN {X 0,Y 585.179,Z 847.637,A -85,B 0,C 180,E1 -8765.555,E2 -8765.555} C_VEL
LIN {X 0,Y 587.18,Z 825.79,A -85,B 0,C 180,E1 -8766.381,E2 -8766.381} C_VEL
LIN {X 0,Y 589.127,Z 802.224,A -85,B 0,C 180,E1 -8767.105,E2 -8767.105} C_VEL
LIN {X 0,Y 590.595,Z 778.451,A -85,B 0,C 180,E1 -8767.648,E2 -8767.648} C_VEL
LIN {X 0,Y 591.557,Z 755.977,A -85,B 0,C 180,E1 -8768.027,E2 -8768.027} C_VEL
LIN {X 0,Y 597.261,Z 506.994,A -85,B 0,C 180,E1 -8771.375,E2 -8771.375} C_VEL
LIN {X 0,Y 599.18,Z 421.264,A -85,B 0,C 180,E1 -8772.552,E2 -8772.552} C_VEL
LIN {X 0,Y 598.222,Z 418.74,A -85,B 0,C 180,E1 -8772.674,E2 -8772.674} C_VEL
LIN {X 0,Y 584.047,Z 394.647,A -85,B 0,C 180,E1 -8774.323,E2 -8774.323} C_VEL
LIN {X 0,Y 570.279,Z 372.684,A -85,B 0,C 180,E1 -8776.027,E2 -8776.027} C_VEL
LIN {X 0,Y 564.417,Z 358.728,A -85,B 0,C 180,E1 -8778.097,E2 -8778.097} C_VEL
LIN {X 0,Y 561.425,Z 351.294,A -85,B 0,C 180,E1 -8779.257,E2 -8779.257} C_VEL
LIN {X 0,Y 561.384,Z 351.292,A -85,B 0,C 180,E1 -8782.344,E2 -8782.344} C_VEL
LIN {X 0,Y 561.388,Z 351.287,A -85,B 0,C 180,E1 -8785.748,E2 -8785.748} C_VEL
LIN {X 0,Y 561.409,Z 351.284,A -85,B 0,C 180,E1 -8788.783,E2 -8788.783} C_VEL
LIN {X 0,Y 561.381,Z 351.287,A -85,B 0,C 180,E1 -8792.067,E2 -8792.067} C_VEL
LIN {X 0,Y 561.443,Z 351.291,A -85,B 0,C 180,E1 -8795.268,E2 -8795.268} C_VEL
LIN {X 0,Y 561.38,Z 351.299,A -85,B 0,C 180,E1 -8798.475,E2 -8798.475} C_VEL
LIN {X 0,Y 561.414,Z 351.282,A -85,B 0,C 180,E1 -8801.732,E2 -8801.732} C_VEL
LIN {X 0,Y 561.395,Z 351.288,A -85,B 0,C 180,E1 -8804.872,E2 -8804.872} C_VEL
LIN {X 0,Y 561.389,Z 351.3,A -85,B 0,C 180,E1 -8808.181,E2 -8808.181} C_VEL
LIN {X 0,Y 561.435,Z 351.276,A -85,B 0,C 180,E1 -8811.396,E2 -8811.396} C_VEL
LIN {X 0,Y 561.379,Z 351.288,A -85,B 0,C 180,E1 -8814.583,E2 -8814.583} C_VEL
LIN {X 0,Y 561.432,Z 351.297,A -85,B 0,C 180,E1 -8817.857,E2 -8817.857} C_VEL
LIN {X 0,Y 561.381,Z 351.274,A -85,B 0,C 180,E1 -8820.919,E2 -8820.919} C_VEL
LIN {X 0,Y 561.399,Z 351.293,A -85,B 0,C 180,E1 -8824.29,E2 -8824.29} C_VEL
LIN {X 0,Y 561.405,Z 351.288,A -85,B 0,C 180,E1 -8827.368,E2 -8827.368} C_VEL
LIN {X 0,Y 561.382,Z 351.278,A -85,B 0,C 180,E1 -8830.675,E2 -8830.675} C_VEL
LIN {X 0,Y 561.45,Z 351.297,A -85,B 0,C 180,E1 -8833.93,E2 -8833.93} C_VEL
LIN {X 0,Y 561.382,Z 351.29,A -85,B 0,C 180,E1 -8837.091,E2 -8837.091} C_VEL
LIN {X 0,Y 561.424,Z 351.279,A -85,B 0,C 180,E1 -8840.322,E2 -8840.322} C_VEL
LIN {X 0,Y 561.392,Z 351.299,A -85,B 0,C 180,E1 -8843.402,E2 -8843.402} C_VEL
LIN {X 0,Y 561.393,Z 351.3,A -85,B 0,C 180,E1 -8846.833,E2 -8846.833} C_VEL
LIN {X 0,Y 561.425,Z 351.278,A -85,B 0,C 180,E1 -8849.913,E2 -8849.913} C_VEL
LIN {X 0,Y 561.382,Z 351.284,A -85,B 0,C 180,E1 -8853.162,E2 -8853.162} C_VEL
LIN {X 0,Y 561.44,Z 351.284,A -85,B 0,C 180,E1 -8856.391,E2 -8856.391} C_VEL
LIN {X 0,Y 561.385,Z 351.292,A -85,B 0,C 180,E1 -8859.536,E2 -8859.536} C_VEL
LIN {X 0,Y 561.413,Z 351.266,A -85,B 0,C 180,E1 -8862.796,E2 -8862.796} C_VEL
LIN {X 0,Y 561.416,Z 351.4,A -85,B 0,C 180,E1 -8865.029,E2 -8865.029} C_VEL
LIN {X 0,Y 561.764,Z 352.877,A -85,B 0,C 180,E1 -8865.16,E2 -8865.16} C_VEL
LIN {X 0,Y 563.667,Z 355.936,A -85,B 0,C 180,E1 -8865.416,E2 -8865.416} C_VEL
LIN {X 0,Y 565.182,Z 357.543,A -85,B 0,C 180,E1 -8865.604,E2 -8865.604} C_VEL
LIN {X 0,Y 567.902,Z 361.521,A -85,B 0,C 180,E1 -8865.955,E2 -8865.955} C_VEL
LIN {X 0,Y 579.907,Z 379.342,A -85,B 0,C 180,E1 -8867.449,E2 -8867.449} C_VEL
LIN {X 0,Y 590.434,Z 396.155,A -85,B 0,C 180,E1 -8868.701,E2 -8868.701} C_VEL
LIN {X 0,Y 599.337,Z 411.062,A -85,B 0,C 180,E1 -8869.718,E2 -8869.718} C_VEL
LIN {X 0,Y 594.323,Z 621.871,A -85,B 0,C 180,E1 -8872.571,E2 -8872.571} C_VEL
LIN {X 0,Y 593.377,Z 629.565,A -85,B 0,C 180,E1 -8872.615,E2 -8872.615} C_VEL
LIN {X 0,Y 588.018,Z 650.1,A -85,B 0,C 180,E1 -8872.509,E2 -8872.509} C_VEL
LIN {X 0,Y 587.273,Z 656.704,A -85,B 0,C 180,E1 -8872.552,E2 -8872.552} C_VEL
LIN {X 0,Y 585.108,Z 741.247,A -85,B 0,C 180,E1 -8873.716,E2 -8873.716} C_VEL
LIN {X 0,Y 583.771,Z 766.42,A -85,B 0,C 180,E1 -8874.229,E2 -8874.229} C_VEL
LIN {X 0,Y 582.282,Z 787.179,A -85,B 0,C 180,E1 -8874.793,E2 -8874.793} C_VEL
LIN {X 0,Y 580.17,Z 811.758,A -85,B 0,C 180,E1 -8875.643,E2 -8875.643} C_VEL
LIN {X 0,Y 578.055,Z 832.103,A -85,B 0,C 180,E1 -8876.51,E2 -8876.51} C_VEL
LIN {X 0,Y 575.616,Z 853.587,A -85,B 0,C 180,E1 -8877.589,E2 -8877.589} C_VEL
LIN {X 0,Y 572.808,Z 875.188,A -85,B 0,C 180,E1 -8878.889,E2 -8878.889} C_VEL
LIN {X 0,Y 570.082,Z 895.415,A -85,B 0,C 180,E1 -8880.298,E2 -8880.298} C_VEL
LIN {X 0,Y 567.3,Z 914.704,A -85,B 0,C 180,E1 -8881.87,E2 -8881.87} C_VEL
LIN {X 0,Y 564.872,Z 931.192,A -85,B 0,C 180,E1 -8883.395,E2 -8883.395} C_VEL
LIN {X 0,Y 562.083,Z 950.048,A -85,B 0,C 180,E1 -8885.401,E2 -8885.401} C_VEL
LIN {X 0,Y 559.944,Z 964.791,A -85,B 0,C 180,E1 -8887.201,E2 -8887.201} C_VEL
LIN {X 0,Y 557.643,Z 981.381,A -85,B 0,C 180,E1 -8889.534,E2 -8889.534} C_VEL
LIN {X 0,Y 556.042,Z 993.781,A -85,B 0,C 180,E1 -8891.549,E2 -8891.549} C_VEL
LIN {X 0,Y 554.51,Z 1007.231,A -85,B 0,C 180,E1 -8894.092,E2 -8894.092} C_VEL
LIN {X 0,Y 553.567,Z 1016.753,A -85,B 0,C 180,E1 -8896.206,E2 -8896.206} C_VEL
LIN {X 0,Y 552.795,Z 1026.378,A -85,B 0,C 180,E1 -8898.735,E2 -8898.735} C_VEL
LIN {X 0,Y 552.35,Z 1033.227,A -85,B 0,C 180,E1 -8900.939,E2 -8900.939} C_VEL
LIN {X 0,Y 552.085,Z 1039.323,A -85,B 0,C 180,E1 -8903.344,E2 -8903.344} C_VEL
LIN {X 0,Y 551.964,Z 1043.913,A -85,B 0,C 180,E1 -8905.845,E2 -8905.845} C_VEL
LIN {X 0,Y 551.926,Z 1046.697,A -85,B 0,C 180,E1 -8908.027,E2 -8908.027} C_VEL
LIN {X 0,Y 551.907,Z 1048.478,A -85,B 0,C 180,E1 -8910.623,E2 -8910.623} C_VEL
LIN {X 0,Y 551.906,Z 1048.598,A -85,B 0,C 180,E1 -8912.908,E2 -8912.908} C_VEL
LIN {X 0,Y 551.915,Z 1047.498,A -85,B 0,C 180,E1 -8915.197,E2 -8915.197} C_VEL
LIN {X 0,Y 551.945,Z 1044.574,A -85,B 0,C 180,E1 -8917.809,E2 -8917.809} C_VEL
LIN {X 0,Y 552.022,Z 1040.994,A -85,B 0,C 180,E1 -8919.909,E2 -8919.909} C_VEL
LIN {X 0,Y 552.247,Z 1035.536,A -85,B 0,C 180,E1 -8922.336,E2 -8922.336} C_VEL
LIN {X 0,Y 552.659,Z 1028.281,A -85,B 0,C 180,E1 -8924.78,E2 -8924.78} C_VEL
LIN {X 0,Y 553.283,Z 1020.145,A -85,B 0,C 180,E1 -8927.057,E2 -8927.057} C_VEL
LIN {X 0,Y 554.253,Z 1009.629,A -85,B 0,C 180,E1 -8929.496,E2 -8929.496} C_VEL
LIN {X 0,Y 555.467,Z 998.753,A -85,B 0,C 180,E1 -8931.655,E2 -8931.655} C_VEL
LIN {X 0,Y 557.208,Z 984.751,A -85,B 0,C 180,E1 -8934.038,E2 -8934.038} C_VEL
LIN {X 0,Y 559.009,Z 971.523,A -85,B 0,C 180,E1 -8935.991,E2 -8935.991} C_VEL
LIN {X 0,Y 561.449,Z 954.593,A -85,B 0,C 180,E1 -8938.169,E2 -8938.169} C_VEL
LIN {X 0,Y 563.739,Z 939.212,A -85,B 0,C 180,E1 -8939.894,E2 -8939.894} C_VEL
LIN {X 0,Y 566.545,Z 920.579,A -85,B 0,C 180,E1 -8941.731,E2 -8941.731} C_VEL
LIN {X 0,Y 569.193,Z 902.626,A -85,B 0,C 180,E1 -8943.261,E2 -8943.261} C_VEL
LIN {X 0,Y 572.136,Z 882.347,A -85,B 0,C 180,E1 -8944.775,E2 -8944.775} C_VEL
LIN {X 0,Y 574.829,Z 861.887,A -85,B 0,C 180,E1 -8946.072,E2 -8946.072} C_VEL
LIN {X 0,Y 577.425,Z 840.954,A -85,B 0,C 180,E1 -8947.22,E2 -8947.22} C_VEL
LIN {X 0,Y 579.913,Z 818.416,A -85,B 0,C 180,E1 -8948.242,E2 -8948.242} C_VEL
LIN {X 0,Y 581.859,Z 798.04,A -85,B 0,C 180,E1 -8949.015,E2 -8949.015} C_VEL
LIN {X 0,Y 583.902,Z 772.802,A -85,B 0,C 180,E1 -8949.773,E2 -8949.773} C_VEL
LIN {X 0,Y 585.175,Z 752.148,A -85,B 0,C 180,E1 -8950.244,E2 -8950.244} C_VEL
LIN {X 0,Y 586.212,Z 727.492,A -85,B 0,C 180,E1 -8950.658,E2 -8950.658} C_VEL
LIN {X 0,Y 592.735,Z 474.327,A -85,B 0,C 180,E1 -8954.122,E2 -8954.122} C_VEL
LIN {X 0,Y 594.185,Z 414.117,A -85,B 0,C 180,E1 -8954.973,E2 -8954.973} C_VEL
LIN {X 0,Y 580.889,Z 392.482,A -85,B 0,C 180,E1 -8956.622,E2 -8956.622} C_VEL
LIN {X 0,Y 568.738,Z 374.274,A -85,B 0,C 180,E1 -8958.216,E2 -8958.216} C_VEL
LIN {X 0,Y 563.794,Z 367.478,A -85,B 0,C 180,E1 -8958.888,E2 -8958.888} C_VEL
LIN {X 0,Y 560.388,Z 362.809,A -85,B 0,C 180,E1 -8959.363,E2 -8959.363} C_VEL
LIN {X 0,Y 557.686,Z 358.97,A -85,B 0,C 180,E1 -8959.75,E2 -8959.75} C_VEL
LIN {X 0,Y 556.886,Z 357.84,A -85,B 0,C 180,E1 -8959.865,E2 -8959.865} C_VEL
LIN {X 0,Y 554.43,Z 355.202,A -85,B 0,C 180,E1 -8960.208,E2 -8960.208} C_VEL
LIN {X 0,Y 553.443,Z 352.256,A -85,B 0,C 180,E1 -8960.426,E2 -8960.426} C_VEL
LIN {X 0,Y 553.49,Z 352.239,A -85,B 0,C 180,E1 -8963.534,E2 -8963.534} C_VEL
LIN {X 0,Y 553.443,Z 352.291,A -85,B 0,C 180,E1 -8966.809,E2 -8966.809} C_VEL
LIN {X 0,Y 553.484,Z 352.286,A -85,B 0,C 180,E1 -8970.128,E2 -8970.128} C_VEL
LIN {X 0,Y 553.454,Z 352.29,A -85,B 0,C 180,E1 -8973.186,E2 -8973.186} C_VEL
LIN {X 0,Y 553.452,Z 352.289,A -85,B 0,C 180,E1 -8976.603,E2 -8976.603} C_VEL
LIN {X 0,Y 553.488,Z 352.282,A -85,B 0,C 180,E1 -8979.705,E2 -8979.705} C_VEL
LIN {X 0,Y 553.441,Z 352.282,A -85,B 0,C 180,E1 -8982.981,E2 -8982.981} C_VEL
LIN {X 0,Y 553.5,Z 352.269,A -85,B 0,C 180,E1 -8986.204,E2 -8986.204} C_VEL
LIN {X 0,Y 553.446,Z 352.281,A -85,B 0,C 180,E1 -8989.381,E2 -8989.381} C_VEL
LIN {X 0,Y 553.451,Z 352.286,A -85,B 0,C 180,E1 -8992.839,E2 -8992.839} C_VEL
LIN {X 0,Y 553.492,Z 352.285,A -85,B 0,C 180,E1 -8996.064,E2 -8996.064} C_VEL
LIN {X 0,Y 553.439,Z 352.277,A -85,B 0,C 180,E1 -8999.275,E2 -8999.275} C_VEL
LIN {X 0,Y 553.494,Z 352.267,A -85,B 0,C 180,E1 -9002.485,E2 -9002.485} C_VEL
LIN {X 0,Y 553.448,Z 352.291,A -85,B 0,C 180,E1 -9005.703,E2 -9005.703} C_VEL
LIN {X 0,Y 553.449,Z 352.288,A -85,B 0,C 180,E1 -9009.148,E2 -9009.148} C_VEL
LIN {X 0,Y 553.498,Z 352.273,A -85,B 0,C 180,E1 -9012.414,E2 -9012.414} C_VEL
LIN {X 0,Y 553.439,Z 352.27,A -85,B 0,C 180,E1 -9015.643,E2 -9015.643} C_VEL
LIN {X 0,Y 553.485,Z 352.268,A -85,B 0,C 180,E1 -9018.867,E2 -9018.867} C_VEL
LIN {X 0,Y 553.453,Z 352.287,A -85,B 0,C 180,E1 -9022.058,E2 -9022.058} C_VEL
LIN {X 0,Y 553.447,Z 352.289,A -85,B 0,C 180,E1 -9025.467,E2 -9025.467} C_VEL
LIN {X 0,Y 553.509,Z 352.286,A -85,B 0,C 180,E1 -9028.719,E2 -9028.719} C_VEL
LIN {X 0,Y 553.44,Z 352.29,A -85,B 0,C 180,E1 -9031.882,E2 -9031.882} C_VEL
LIN {X 0,Y 553.483,Z 352.288,A -85,B 0,C 180,E1 -9035.19,E2 -9035.19} C_VEL
LIN {X 0,Y 553.454,Z 352.291,A -85,B 0,C 180,E1 -9038.364,E2 -9038.364} C_VEL
LIN {X 0,Y 553.479,Z 352.358,A -85,B 0,C 180,E1 -9039.384,E2 -9039.384} C_VEL
LIN {X 0,Y 554.665,Z 355.655,A -85,B 0,C 180,E1 -9039.923,E2 -9039.923} C_VEL
LIN {X 0,Y 558.806,Z 364.624,A -85,B 0,C 180,E1 -9041.457,E2 -9041.457} C_VEL
LIN {X 0,Y 562.281,Z 372.587,A -85,B 0,C 180,E1 -9042.703,E2 -9042.703} C_VEL
LIN {X 0,Y 574.651,Z 391.348,A -85,B 0,C 180,E1 -9044.385,E2 -9044.385} C_VEL
LIN {X 0,Y 587.888,Z 412.893,A -85,B 0,C 180,E1 -9046.079,E2 -9046.079} C_VEL
LIN {X 0,Y 594.346,Z 424.545,A -85,B 0,C 180,E1 -9046.879,E2 -9046.879} C_VEL
LIN {X 0,Y 587.539,Z 685.487,A -85,B 0,C 180,E1 -9050.462,E2 -9050.462} C_VEL
LIN {X 0,Y 585.395,Z 765.84,A -85,B 0,C 180,E1 -9051.577,E2 -9051.577} C_VEL
LIN {X 0,Y 583.856,Z 791.505,A -85,B 0,C 180,E1 -9052.093,E2 -9052.093} C_VEL
LIN {X 0,Y 582.157,Z 813.446,A -85,B 0,C 180,E1 -9052.689,E2 -9052.689} C_VEL
LIN {X 0,Y 579.857,Z 838.217,A -85,B 0,C 180,E1 -9053.555,E2 -9053.555} C_VEL
LIN {X 0,Y 577.731,Z 857.924,A -85,B 0,C 180,E1 -9054.399,E2 -9054.399} C_VEL
LIN {X 0,Y 575.077,Z 880.382,A -85,B 0,C 180,E1 -9055.532,E2 -9055.532} C_VEL
LIN {X 0,Y 572.309,Z 901.331,A -85,B 0,C 180,E1 -9056.795,E2 -9056.795} C_VEL
LIN {X 0,Y 569.514,Z 921.819,A -85,B 0,C 180,E1 -9058.217,E2 -9058.217} C_VEL
LIN {X 0,Y 566.635,Z 941.805,A -85,B 0,C 180,E1 -9059.844,E2 -9059.844} C_VEL
LIN {X 0,Y 564.042,Z 959.907,A -85,B 0,C 180,E1 -9061.519,E2 -9061.519} C_VEL
LIN {X 0,Y 561.436,Z 977.937,A -85,B 0,C 180,E1 -9063.447,E2 -9063.447} C_VEL
LIN {X 0,Y 559.365,Z 993.012,A -85,B 0,C 180,E1 -9065.274,E2 -9065.274} C_VEL
LIN {X 0,Y 557.245,Z 1009.251,A -85,B 0,C 180,E1 -9067.532,E2 -9067.532} C_VEL
LIN {X 0,Y 555.717,Z 1022.031,A -85,B 0,C 180,E1 -9069.57,E2 -9069.57} C_VEL
LIN {X 0,Y 554.313,Z 1035.345,A -85,B 0,C 180,E1 -9072.034,E2 -9072.034} C_VEL
LIN {X 0,Y 553.459,Z 1044.756,A -85,B 0,C 180,E1 -9074.061,E2 -9074.061} C_VEL
LIN {X 0,Y 552.749,Z 1054.477,A -85,B 0,C 180,E1 -9076.505,E2 -9076.505} C_VEL
LIN {X 0,Y 552.313,Z 1061.979,A -85,B 0,C 180,E1 -9078.831,E2 -9078.831} C_VEL
LIN {X 0,Y 552.061,Z 1068.073,A -85,B 0,C 180,E1 -9081.144,E2 -9081.144} C_VEL
LIN {X 0,Y 551.95,Z 1072.982,A -85,B 0,C 180,E1 -9083.656,E2 -9083.656} C_VEL
LIN {X 0,Y 551.916,Z 1075.818,A -85,B 0,C 180,E1 -9085.74,E2 -9085.74} C_VEL
LIN {X 0,Y 551.907,Z 1077.7,A -85,B 0,C 180,E1 -9088.027,E2 -9088.027} C_VEL
LIN {X 0,Y 551.899,Z 1078.132,A -85,B 0,C 180,E1 -9090.519,E2 -9090.519} C_VEL
LIN {X 0,Y 551.91,Z 1077.216,A -85,B 0,C 180,E1 -9092.7,E2 -9092.7} C_VEL
LIN {X 0,Y 551.933,Z 1074.893,A -85,B 0,C 180,E1 -9095.093,E2 -9095.093} C_VEL
LIN {X 0,Y 551.985,Z 1070.925,A -85,B 0,C 180,E1 -9097.494,E2 -9097.494} C_VEL
LIN {X 0,Y 552.143,Z 1066.011,A -85,B 0,C 180,E1 -9099.696,E2 -9099.696} C_VEL
LIN {X 0,Y 552.484,Z 1058.767,A -85,B 0,C 180,E1 -9102.231,E2 -9102.231} C_VEL
LIN {X 0,Y 552.991,Z 1050.86,A -85,B 0,C 180,E1 -9104.449,E2 -9104.449} C_VEL
LIN {X 0,Y 553.802,Z 1041.052,A -85,B 0,C 180,E1 -9106.791,E2 -9106.791} C_VEL
LIN {X 0,Y 554.932,Z 1029.263,A -85,B 0,C 180,E1 -9109.143,E2 -9109.143} C_VEL
LIN {X 0,Y 556.317,Z 1016.916,A -85,B 0,C 180,E1 -9111.288,E2 -9111.288} C_VEL
LIN {X 0,Y 558.197,Z 1001.827,A -85,B 0,C 180,E1 -9113.544,E2 -9113.544} C_VEL
LIN {X 0,Y 560.083,Z 987.69,A -85,B 0,C 180,E1 -9115.399,E2 -9115.399} C_VEL
LIN {X 0,Y 562.679,Z 969.137,A -85,B 0,C 180,E1 -9117.518,E2 -9117.518} C_VEL
LIN {X 0,Y 564.952,Z 953.042,A -85,B 0,C 180,E1 -9119.125,E2 -9119.125} C_VEL
LIN {X 0,Y 567.91,Z 932.216,A -85,B 0,C 180,E1 -9120.938,E2 -9120.938} C_VEL
LIN {X 0,Y 570.445,Z 913.895,A -85,B 0,C 180,E1 -9122.318,E2 -9122.318} C_VEL
LIN {X 0,Y 573.323,Z 892.216,A -85,B 0,C 180,E1 -9123.737,E2 -9123.737} C_VEL
LIN {X 0,Y 575.838,Z 871.262,A -85,B 0,C 180,E1 -9124.9,E2 -9124.9} C_VEL
LIN {X 0,Y 578.364,Z 849.264,A -85,B 0,C 180,E1 -9125.94,E2 -9125.94} C_VEL
LIN {X 0,Y 580.57,Z 826.283,A -85,B 0,C 180,E1 -9126.823,E2 -9126.823} C_VEL
LIN {X 0,Y 582.501,Z 803.812,A -85,B 0,C 180,E1 -9127.525,E2 -9127.525} C_VEL
LIN {X 0,Y 584.13,Z 779.377,A -85,B 0,C 180,E1 -9128.1,E2 -9128.1} C_VEL
LIN {X 0,Y 585.129,Z 757.488,A -85,B 0,C 180,E1 -9128.478,E2 -9128.478} C_VEL
LIN {X 0,Y 591.025,Z 513.048,A -85,B 0,C 180,E1 -9131.798,E2 -9131.798} C_VEL
LIN {X 0,Y 593.157,Z 423.688,A -85,B 0,C 180,E1 -9133.032,E2 -9133.032} C_VEL
LIN {X 0,Y 578.927,Z 399.379,A -85,B 0,C 180,E1 -9134.724,E2 -9134.724} C_VEL
LIN {X 0,Y 565.486,Z 377.953,A -85,B 0,C 180,E1 -9136.419,E2 -9136.419} C_VEL
LIN {X 0,Y 561.718,Z 372.03,A -85,B 0,C 180,E1 -9136.948,E2 -9136.948} C_VEL
LIN {X 0,Y 554.96,Z 356.032,A -85,B 0,C 180,E1 -9139.426,E2 -9139.426} C_VEL
LIN {X 0,Y 553.473,Z 352.517,A -85,B 0,C 180,E1 -9139.995,E2 -9139.995} C_VEL
LIN {X 0,Y 553.493,Z 352.272,A -85,B 0,C 180,E1 -9142.888,E2 -9142.888} C_VEL
LIN {X 0,Y 553.44,Z 352.278,A -85,B 0,C 180,E1 -9146.189,E2 -9146.189} C_VEL
LIN {X 0,Y 553.479,Z 352.271,A -85,B 0,C 180,E1 -9149.493,E2 -9149.493} C_VEL
LIN {X 0,Y 553.448,Z 352.27,A -85,B 0,C 180,E1 -9152.568,E2 -9152.568} C_VEL
LIN {X 0,Y 553.445,Z 352.273,A -85,B 0,C 180,E1 -9156.015,E2 -9156.015} C_VEL
LIN {X 0,Y 553.496,Z 352.286,A -85,B 0,C 180,E1 -9159.152,E2 -9159.152} C_VEL
LIN {X 0,Y 553.441,Z 352.287,A -85,B 0,C 180,E1 -9162.439,E2 -9162.439} C_VEL
LIN {X 0,Y 553.491,Z 352.264,A -85,B 0,C 180,E1 -9165.671,E2 -9165.671} C_VEL
LIN {X 0,Y 553.452,Z 352.286,A -85,B 0,C 180,E1 -9168.854,E2 -9168.854} C_VEL
LIN {X 0,Y 553.447,Z 352.29,A -85,B 0,C 180,E1 -9172.317,E2 -9172.317} C_VEL
LIN {X 0,Y 553.49,Z 352.262,A -85,B 0,C 180,E1 -9175.441,E2 -9175.441} C_VEL
LIN {X 0,Y 553.441,Z 352.288,A -85,B 0,C 180,E1 -9178.654,E2 -9178.654} C_VEL
LIN {X 0,Y 553.496,Z 352.266,A -85,B 0,C 180,E1 -9181.863,E2 -9181.863} C_VEL
LIN {X 0,Y 553.448,Z 352.277,A -85,B 0,C 180,E1 -9185.079,E2 -9185.079} C_VEL
LIN {X 0,Y 553.451,Z 352.29,A -85,B 0,C 180,E1 -9188.519,E2 -9188.519} C_VEL
LIN {X 0,Y 553.495,Z 352.26,A -85,B 0,C 180,E1 -9191.779,E2 -9191.779} C_VEL
LIN {X 0,Y 553.442,Z 352.281,A -85,B 0,C 180,E1 -9194.973,E2 -9194.973} C_VEL
LIN {X 0,Y 553.493,Z 352.285,A -85,B 0,C 180,E1 -9198.212,E2 -9198.212} C_VEL
LIN {X 0,Y 553.452,Z 352.269,A -85,B 0,C 180,E1 -9201.404,E2 -9201.404} C_VEL
LIN {X 0,Y 553.453,Z 352.27,A -85,B 0,C 180,E1 -9204.78,E2 -9204.78} C_VEL
LIN {X 0,Y 553.502,Z 352.284,A -85,B 0,C 180,E1 -9208.014,E2 -9208.014} C_VEL
LIN {X 0,Y 553.446,Z 352.29,A -85,B 0,C 180,E1 -9211.233,E2 -9211.233} C_VEL
LIN {X 0,Y 553.487,Z 352.281,A -85,B 0,C 180,E1 -9214.535,E2 -9214.535} C_VEL
LIN {X 0,Y 553.461,Z 352.285,A -85,B 0,C 180,E1 -9217.767,E2 -9217.767} C_VEL
LIN {X 0,Y 553.453,Z 352.292,A -85,B 0,C 180,E1 -9221.119,E2 -9221.119} C_VEL
LIN {X 0,Y 553.516,Z 352.422,A -85,B 0,C 180,E1 -9224.253,E2 -9224.253} C_VEL
LIN {X 0,Y 554.737,Z 355.613,A -85,B 0,C 180,E1 -9224.448,E2 -9224.448} C_VEL
LIN {X 0,Y 557.304,Z 358.568,A -85,B 0,C 180,E1 -9224.784,E2 -9224.784} C_VEL
LIN {X 0,Y 560.041,Z 362.58,A -85,B 0,C 180,E1 -9225.152,E2 -9225.152} C_VEL
LIN {X 0,Y 567.608,Z 373.212,A -85,B 0,C 180,E1 -9226.132,E2 -9226.132} C_VEL
LIN {X 0,Y 581.618,Z 394.667,A -85,B 0,C 180,E1 -9227.868,E2 -9227.868} C_VEL
LIN {X 0,Y 593.291,Z 414.33,A -85,B 0,C 180,E1 -9229.247,E2 -9229.247} C_VEL
LIN {X 0,Y 587.273,Z 656.704,A -85,B 0,C 180,E1 -9232.552,E2 -9232.552} C_VEL
